// TIA Portal project "Diplomski_rad" (V16)

(* hardware
DEVICE "S7-1200 station_2"  S7-1200 Station
   slot 0: "Rack_0"  S7-1200 Rack  Rack  V1.0
   slot 1: "PLC_1"  CPU 1215C DC/DC/DC  6ES7 215-1AG40-0XB0  V4.4
DEVICE "HMI_1"  KTP700 Basic PN
   slot 0: "HMI_1"  KTP700 Basic PN  6AV2 123-2GB03-0AX0  16.0.0.0
   slot 1: "HMI_RT_1"  KTP700 Basic PN  6AV2 123-2GB03-0AX0  16.0.0.0
   slot 5: "HMI_1.IE_CP_1"  PROFINET Interface  16.0.0.0
      slot 1: "PROFINET Interface_1"  PROFINET Interface
         slot 1: "Port_1"  Port
DEVICE "SCALANCE X005"  SCALANCE X-Station
   slot 0: "SCALANCE X rack"  Rail
   slot 0: "Switch_1"  6GK5 005-0BA00-1AB2  V1.0
DEVICE "GSD device_1"  GSD.Device.PN
   slot 0: "Rack"  Rack  V1.0
   slot 0: "EX260-SPN"  EX260 SPN 1/2  EX260-SPN
      slot 0: "EX260 SPN 1/2"  EX260 SPN 1/2
      slot 1: "Interface"  Interface
         slot 1: "Port 1 - RJ45"  Port 1 - RJ45
         slot 2: "Port 2 - RJ45"  Port 2 - RJ45
      slot 1: "  4 byte  Output_1"    4 byte  Output
         slot 0: "  4 byte  Output"    4 byte  Output
DEVICE "ET 200SP station_1"  ET 200SP-Station
   slot 0: "Rack_0"  Rack  6ES5 710-8MAx1
   slot 0: "IO device_1"  IM 155-6 PN/2 HF  6ES7 155-6AU01-0CN0  V4.2
   slot 1: "DI 8x24VDC HF_1"  DI 8x24VDC HF  6ES7 131-6BF00-0CA0  V2.0
      slot 1: "DI 8x24VDC HF_1"  DI 8x24VDC HF
   slot 2: "DI 8x24VDC HF_2"  DI 8x24VDC HF  6ES7 131-6BF00-0CA0  V2.0
      slot 1: "DI 8x24VDC HF_2"  DI 8x24VDC HF
   slot 3: "DQ 8x24VDC/0.5A HF_1"  DQ 8x24VDC/0.5A HF  6ES7 132-6BF00-0CA0  V2.0
      slot 1: "DQ 8x24VDC/0.5A HF_1"  DQ 8x24VDC/0.5A HF
   slot 4: "DQ 8x24VDC/0.5A HF_2"  DQ 8x24VDC/0.5A HF  6ES7 132-6BF00-0CA0  V2.0
      slot 1: "DQ 8x24VDC/0.5A HF_2"  DQ 8x24VDC/0.5A HF
   slot 5: "AI 4xU/I 2-wire ST_1"  AI 4xU/I 2-wire ST  6ES7 134-6HD01-0BA1  V2.0
      slot 1: "AI 4xU/I 2-wire ST_1"  AI 4xU/I 2-wire ST
   slot 6: "AQ 2xU/I HF_1"  AQ 2xU/I HF  6ES7 135-6HB00-0CA1  V1.0
      slot 1: "AQ 2xU/I HF_1"  AQ 2xU/I HF
   slot 7: "TM Timer DIDQ 10x24V_1"  TM Timer DIDQ 10x24V  6ES7 138-6CG00-0BA0  V1.0
      slot 1: "TM Timer DIDQ 10x24V_1"  TM Timer DIDQ 10x24V
   slot 8: "Server module_1"  Server module  6ES7 193-6PA00-0AA0  V1.1
      slot 1: "Server module_1"  Server module
   slot 127: "BA 2xRJ45"  BA 2xRJ45  6ES7 193-6AR00-0AA0  V0.0
      slot 1: "Port_1"  X1 P1 R  6ES7 193-6AR00-0AA0  V0.0
      slot 2: "Port_2"  X1 P2 R  6ES7 193-6AR00-0AA0  V0.0
*)

// ===== PLC "PLC_1"  CPU 1215C DC/DC/DC =====

VAR_GLOBAL   // PLC tag table "Default tag table"
   "Tag_1" AT %M0.0 : Bool;
   "Tag_2" AT %M0.1 : Bool;
   "Tag_3" AT %M0.2 : Bool;
   "Tag_4" AT %M0.3 : Bool;
   "Tag_5" AT %M0.4 : Bool;
END_VAR

VAR_GLOBAL   // PLC tag table "PLC I/O"
   "izlaz1" AT %Q0.0 : Bool;   // PTO_motor_1
   "izlaz2" AT %Q0.1 : Bool;   // Enable_motor_1
   "izlaz3" AT %Q0.2 : Bool;   // Direction_motor_1
   "izlaz4" AT %Q0.3 : Bool;   // PTO_motor_2
   "izlaz5" AT %Q0.4 : Bool;   // Enable_motor_2
   "izlaz6" AT %Q0.5 : Bool;   // Direction_motor_2
   "izlaz7" AT %Q0.6 : Bool;
   "izlaz8" AT %Q0.7 : Bool;
   "ulaz1" AT %I0.0 : Bool;
   "ulaz2" AT %I0.1 : Bool;
   "ulaz3" AT %I0.2 : Bool;   // Home_vodilica_1_(manja)
   "ulaz4" AT %I0.3 : Bool;   // Home_vodilica_2_(veca)
   "ulaz5" AT %I0.4 : Bool;   // HW_limiter_0_vodilica_1
   "ulaz6" AT %I0.5 : Bool;   // HW_limiter_1_vodilica_1
   "ulaz7" AT %I0.6 : Bool;   // HW_limiter_0_vodilica_2
   "ulaz8" AT %I0.7 : Bool;   // HW_limiter_1_vodilica_2
END_VAR

VAR_GLOBAL   // PLC tag table "Distro I/O"
   "Dist_ulaz1" AT %I2.0 : Bool;
   "Dist_ulaz2" AT %I2.1 : Bool;
   "Dist_ulaz3" AT %I2.2 : Bool;
   "Dist_ulaz4" AT %I2.3 : Bool;
   "Dist_ulaz5" AT %I2.4 : Bool;   // Senzor_cilindar_uvučen
   "Dist_ulaz6" AT %I2.5 : Bool;   // Senzor_cilindar_izvučen
   "Dist_ulaz7" AT %I2.6 : Bool;   // Senzor_hvataljka_otvorena
   "Dist_ulaz8" AT %I2.7 : Bool;   // Senzor_hvataljka_zatvorena
   "Dist_izlaz1" AT %Q2.0 : Bool;
   "Dist_izlaz2" AT %Q2.1 : Bool;
   "Dist_izlaz3" AT %Q2.2 : Bool;
   "Dist_izlaz4" AT %Q2.3 : Bool;
   "Dist_izlaz5" AT %Q2.4 : Bool;
   "Dist_izlaz6" AT %Q2.5 : Bool;
   "Dist_izlaz7" AT %Q2.6 : Bool;
   "Dist_izlaz8" AT %Q2.7 : Bool;
END_VAR

VAR_GLOBAL   // PLC tag table "Ventili I/O"
   "Ventil_izlaz_1" AT %Q4.0 : Bool;
   "Ventil_izlaz_2" AT %Q4.1 : Bool;
   "Ventil_izlaz_3" AT %Q4.2 : Bool;
   "Ventil_izlaz_4" AT %Q4.3 : Bool;
   "Otvorena_hvataljka" AT %Q4.4 : Bool;
   "Zatvorena_hvataljka" AT %Q4.5 : Bool;
   "Izvučeni_cilindar" AT %Q4.6 : Bool;
   "Uvučeni_cilindar" AT %Q4.7 : Bool;
   "Ventil_izlaz_9" AT %Q5.0 : Bool;
   "Ventil_izlaz_10" AT %Q5.1 : Bool;
   "Ventil_izlaz_11" AT %Q5.2 : Bool;
   "Ventil_izlaz_12" AT %Q5.3 : Bool;
   "Ventil_izlaz_13" AT %Q5.4 : Bool;
   "Ventil_izlaz_14" AT %Q5.5 : Bool;
   "Ventil_izlaz_15" AT %Q5.6 : Bool;
   "Ventil_izlaz_16" AT %Q5.7 : Bool;
   "Ventil_izlaz_17" AT %Q6.0 : Bool;
   "Ventil_izlaz_18" AT %Q6.1 : Bool;
   "Ventil_izlaz_19" AT %Q6.2 : Bool;
   "Ventil_izlaz_20" AT %Q6.3 : Bool;
   "Ventil_izlaz_21" AT %Q6.4 : Bool;
   "Ventil_izlaz_22" AT %Q6.5 : Bool;
   "Ventil_izlaz_23" AT %Q6.6 : Bool;
   "Ventil_izlaz_24" AT %Q6.7 : Bool;
   "Ventil_izlaz_25" AT %Q7.0 : Bool;
   "Ventil_izlaz_26" AT %Q7.1 : Bool;
   "Ventil_izlaz_27" AT %Q7.2 : Bool;
   "Ventil_izlaz_28" AT %Q7.3 : Bool;
   "Ventil_izlaz_29" AT %Q7.4 : Bool;
   "Ventil_izlaz_30" AT %Q7.5 : Bool;
   "Ventil_izlaz_31" AT %Q7.6 : Bool;
   "Ventil_izlaz_32" AT %Q7.7 : Bool;
END_VAR

TYPE "Motor"
   STRUCT
      Uključi_motor : Bool;
      "Potvrdi_error(reset)" : Bool;
      Pokreni_homing : Bool;
      Pokreni_zaustavljanje : Bool;
      Pokreni_izvršavanje_pomaka_apsolutno : Bool;
      Pokreni_izvršavanje_pomaka_relativno : Bool;
      Željena_pozicija : Real;
      Željeni_pomak : Real;
      Trenutna_pozicija : Real;
      Power_Status : Bool;
      Power_Error : Bool;
      "Potvrdi_error(reset)_Izvršeno" : Bool;
      "Potvrdi_error(reset)_Error" : Bool;
      Home_Izvršeno : Bool;
      Home_izvršeno_barem_jednom : Bool;
      Home_Izvršavanje : Bool;
      Home_Error : Bool;
      Halt_Izvršeno : Bool;
      Halt_Error : Bool;
      Pomak_Apsolutno_Izvršeno : Bool;
      Pomak_Apsolutno_U_Tijeku : Bool;
      Pomak_Apsolutno_Error : Bool;
      Pomak_Relativno_izvršeno : Bool;
      Pomak_Relativno_Error : Bool;
      Brzina_Izvršavanje : Bool;
      Brzina_Error : Bool;
   END_STRUCT;
END_TYPE

DATA_BLOCK "Motor_DB"   // DB2
{ S7_Optimized_Access := 'TRUE' }
VERSION : 0.1
   VAR
      "Motor_1_x-os" : "Motor";
      "Motor_2_y-os" : "Motor";
   END_VAR
BEGIN
END_DATA_BLOCK

DATA_BLOCK "Rucno_upravljanje"   // DB3
{ S7_Optimized_Access := 'TRUE' }
VERSION : 0.1
   VAR
      GORE : Bool;
      DOLJE : Bool;
      LIJEVO : Bool;
      DESNO : Bool;
      GD_izvrsavanje : Bool;
      LD_izvrsavanje : Bool;
      GD_brzina : Real := 12.0;
      LD_brzina : Real := 12.0;
   END_VAR
BEGIN
END_DATA_BLOCK

DATA_BLOCK "Pneumatske_komponente"   // DB5
{ S7_Optimized_Access := 'TRUE' }
VERSION : 0.1
   VAR
      Aktivacija_cilindra : Bool;
      Aktivacija_hvataljke : Bool;
   END_VAR
BEGIN
END_DATA_BLOCK

DATA_BLOCK "Paletizacija_DB"   // DB6
{ S7_Optimized_Access := 'TRUE' }
VERSION : 0.1
// stored: InstanceOfName Paletizacija
"Paletizacija"
BEGIN
END_DATA_BLOCK

DATA_BLOCK "Automatsko_upravljanje"   // DB7
{ S7_Optimized_Access := 'TRUE' }
VERSION : 0.1
   VAR
      Automatski_režim : Bool;
      Paletizacija : Bool;
      Kraj_paletizacije : Bool;
      Broj_komada_palete_x : Int := 2;
      Broj_komada_palete_y : Int := 2;
      Pauza : Bool;
      Lokalizacija_objekata_i_sortiranje : Bool;
      Lokalizacija_objekata_x_koordinata : Real;
      Lokalizacija_objekata_y_koordinata : Real;
      Primljeni_podatci : Bool;
      Lokalizacija_objekata_boja : Int;
      Zahtjev_za_poziciju : Bool;
   END_VAR
BEGIN
END_DATA_BLOCK

DATA_BLOCK "Vizija_python"   // DB10
{ S7_Optimized_Access := 'FALSE' }
VERSION : 0.1
   VAR
      Slanje_podataka : Byte;
      Slanje_podataka_stanje : Bool;
      Primanje_podataka : Char;
      Broj_primljenih_podataka : Int := 0;
      Primljeno : Bool;
      Broj : DInt;
      X_koordinata : DInt := 0;
      Y_koordinata : DInt := 0;
      Boja : DInt := 0;
      Broj_razmaka : DInt := 0;
      "Koeficijent_px/mm_x" : Real := 4.9;
      "Koeficijent_px/mm_y" : Real := 4.85;
      Offset_k_s_kamere_x : Real := 0.0;
      Offset_k_s_kamere_y : Real := 47.0;
   END_VAR
BEGIN
END_DATA_BLOCK

DATA_BLOCK "Lokalizacija_objekata_i_sortiranje_DB"   // DB13
{ S7_Optimized_Access := 'TRUE' }
VERSION : 0.1
// stored: InstanceOfName Lokalizacija_objekata_i_sortiranje
"Lokalizacija_objekata_i_sortiranje"
BEGIN
END_DATA_BLOCK

DATA_BLOCK "Motor_upravljanje_DB"   // DB17
{ S7_Optimized_Access := 'TRUE' }
VERSION : 0.1
// stored: InstanceOfName Motor_upravljanje
"Motor_upravljanje"
BEGIN
END_DATA_BLOCK

DATA_BLOCK "Motor_upravljanje_DB_2"   // DB18
{ S7_Optimized_Access := 'TRUE' }
VERSION : 0.1
// stored: InstanceOfName Motor_upravljanje
"Motor_upravljanje"
BEGIN
END_DATA_BLOCK

// folder: System blocks/Program resources

DATA_BLOCK "PLC_1_TCP_DB"   // DB9
{ S7_Optimized_Access := 'TRUE' }
AUTHOR : SIMATIC
FAMILY : MC7Plus
NAME : TC_IP_v4
VERSION : 1.0
// stored: InstanceOfName TCON_IP_v4
"TCON_IP_v4"
BEGIN
   ID := 1;
   InterfaceId := 64;
   LocalPort := 2000;
END_DATA_BLOCK

DATA_BLOCK "Tajmer_za_slanje_poruke"   // DB12
{ S7_Optimized_Access := 'TRUE' }
AUTHOR : Simatic
FAMILY : IEC
NAME : IEC_TMR
VERSION : 1.0
// stored: InstanceOfName IEC_TIMER
"IEC_TIMER"
BEGIN
END_DATA_BLOCK

DATA_BLOCK "IEC_Timer_0_DB_1"   // DB14
{ S7_Optimized_Access := 'TRUE' }
AUTHOR : Simatic
FAMILY : IEC
NAME : IEC_TMR
VERSION : 1.0
// stored: InstanceOfName IEC_TIMER
"IEC_TIMER"
BEGIN
END_DATA_BLOCK

DATA_BLOCK "Tajmer_za_primanje_poruke"   // DB15
{ S7_Optimized_Access := 'TRUE' }
AUTHOR : Simatic
FAMILY : IEC
NAME : IEC_TMR
VERSION : 1.0
// stored: InstanceOfName IEC_TIMER
"IEC_TIMER"
BEGIN
END_DATA_BLOCK

// folder: (top level)

DATA_BLOCK "Axis_1"   // DB1, Motion_DB
{ S7_Optimized_Access := 'TRUE' }
AUTHOR : SIMATIC
FAMILY : BasicMC
NAME : TO_PosAx
VERSION : 7.0
// stored: InstanceOfName TO_PositioningAxis
"TO_PositioningAxis"
BEGIN
   // Axis.DirectionOutputEnabledCU = TRUE
   // Axis.PositionLimitsMax_AddressCU = %I0.5
   // Axis.PositionLimitsMin_AddressCU = %I0.4
   // Axis.PassiveHomingReferencePointSwitch_AddressCU = %I0.2
   // Axis.HomingReferencePointSwitch_AddressCU = %I0.2
   // Axis.LengthUnitNormalized.Distance = 1013
   // Axis.EnableOutput_AddressCU = %Q0.1
   // Axis.OnlinePtoModeCU = 16#0000_0002
   // Axis.SelectedChannel2EnumCU = %Q0.2
   // Axis.SelectedChannel1EnumCU = %Q0.0
   // Pulse.MinDeltaDeltaFrequencyCU = 0.004
   // Pulse.MaxDeltaDeltaFrequencyCU = 1.0E+10
   // Pulse.MinDeltaFrequencyCU = 0.005
   // Pulse.MaxDeltaFrequencyCU = 9.5E+9
   // Pulse.MinFrequencyCU = 1.0
   // Pulse.MaxFrequencyCU = 100000.0
   // Pulse.OutputSourceCU = 16#0000_0000
   // Axis.SelectPTO = 0
END_DATA_BLOCK

DATA_BLOCK "Axis_2"   // DB4, Motion_DB
{ S7_Optimized_Access := 'TRUE' }
AUTHOR : SIMATIC
FAMILY : BasicMC
NAME : TO_PosAx
VERSION : 7.0
// stored: InstanceOfName TO_PositioningAxis
"TO_PositioningAxis"
BEGIN
   // Axis.PositionLimitsMax_AddressCU = %I0.7
   // Axis.PositionLimitsMin_AddressCU = %I0.6
   // Axis.PassiveHomingReferencePointSwitch_AddressCU = %I0.3
   // Axis.HomingReferencePointSwitch_AddressCU = %I0.3
   // Axis.LengthUnitNormalized.Distance = 1013
   // Axis.EnableOutput_AddressCU = %Q0.4
   // Axis.OnlinePtoModeCU = 16#0000_0002
   // Axis.DirectionOutputEnabledCU = TRUE
   // Axis.SelectedChannel2EnumCU = %Q0.5
   // Axis.SelectedChannel1EnumCU = %Q0.3
   // Pulse.MinDeltaDeltaFrequencyCU = 0.004
   // Pulse.MaxDeltaDeltaFrequencyCU = 1.0E+10
   // Pulse.MinDeltaFrequencyCU = 0.005
   // Pulse.MaxDeltaFrequencyCU = 9.5E+9
   // Pulse.MinFrequencyCU = 1.0
   // Pulse.MaxFrequencyCU = 100000.0
   // Pulse.OutputSourceCU = 16#0000_0000
   // Axis.SelectPTO = 1
   // Axis.OnlinePtoIndexCU = 1
END_DATA_BLOCK

FUNCTION_BLOCK "Motor_upravljanje"   // FB1, LAD
{ S7_Optimized_Access := 'TRUE' }
VERSION : 0.1
   VAR_INPUT
      Os : TO_PositioningAxis;
      Uključi_motor : Bool;
      "Potvrdi_error(reset)" : Bool;
      Pokreni_homing : Bool;
      Pokreni_zaustavljanje : Bool;
      Pokreni_izvršavanje_pomaka_apsolutno : Bool;
      Pokreni_izvršavanje_pomaka_relativno : Bool;
      Željena_pozicija : Real;
      Željeni_pomak : Real;
      Izvršavanje_direktno_preko_gumba : Bool;
      Maks_brzina_izvršavanje_preko_gumba : Real;
      Gumb_od_motora : Bool;
      Gumb_prema_motoru : Bool;
   END_VAR
   VAR_OUTPUT
      Trenutna_pozicija : Real;
      Power_Status : Bool;
      Power_Error : Bool;
      "Potvrdi_error(reset)_Izvršeno" : Bool;
      "Potvrdi_error(reset)_Error" : Bool;
      Home_Izvršeno : Bool;
      Home_izvršeno_barem_jednom : Bool;
      Home_izvršavanje : Bool;
      Home_Error : Bool;
      Halt_Izvršeno : Bool;
      Halt_Error : Bool;
      Pomak_Apsolutno_Izvršeno : Bool;
      Pomak_Apsolutno_U_Tijeku : Bool;
      Pomak_Apsolutno_Error : Bool;
      Pomak_Relativno_Izvršeno : Bool;
      Pomak_Relativno_Error : Bool;
      Brzina_Izvršavanje : Bool;
      Brzina_Error : Bool;
   END_VAR
   VAR
      MC_Power_Instance : MC_Power;
      MC_Reset_Instance : MC_Reset;
      MC_Home_Instance : MC_Home;
      MC_Halt_Instance : MC_Halt;
      MC_MoveAbsolute_Instance : MC_MoveAbsolute;
      MC_MoveRelative_Instance : MC_MoveRelative;
      MC_MoveVelocity_Instance : MC_MoveVelocity;
      Provjera_edga : Bool;
   END_VAR
   VAR_TEMP   // added for the SCL form of the ladder/FBD networks
      _w1 : Bool;
   END_VAR
BEGIN

REGION Network 1
   // MC_Power - Uključuje motor, bez njega se ne može pokrenuti
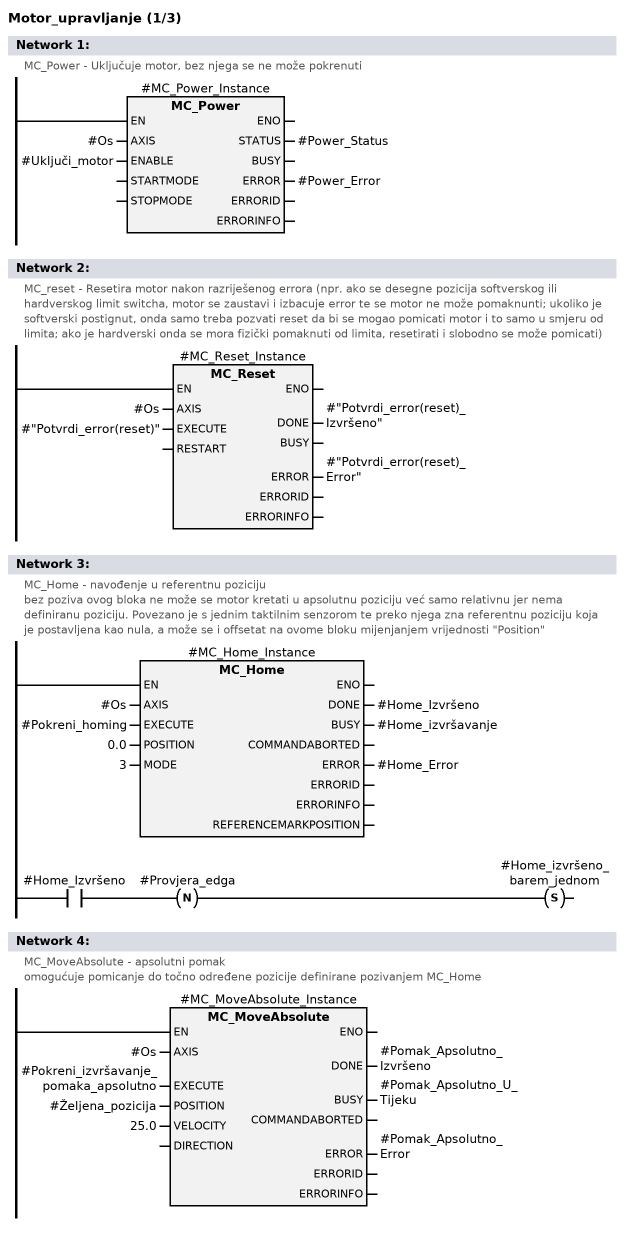
   #MC_Power_Instance(Axis := #Os, Enable := #Uključi_motor, Status => #Power_Status, Error => #Power_Error);   // MC_Power
END_REGION

REGION Network 2
   // MC_reset - Resetira motor nakon razriješenog errora (npr. ako se desegne pozicija softverskog ili hardverskog limit switcha, motor se zaustavi i izbacuje error te se motor ne može pomaknunti; ukoliko je softverski postignut, onda samo treba pozvati reset da bi se mogao pomicati motor i to samo u smjeru od limita; ako je hardverski onda se mora fizički pomaknuti od limita, resetirati i slobodno se može pomicati)
   #MC_Reset_Instance(Axis := #Os,   // MC_Reset
                      Execute := #"Potvrdi_error(reset)",
                      Done => #"Potvrdi_error(reset)_Izvršeno",
                      Error => #"Potvrdi_error(reset)_Error");
END_REGION

REGION Network 3
   // MC_Home - navođenje u referentnu poziciju
   // bez poziva ovog bloka ne može se motor kretati u apsolutnu poziciju već samo relativnu jer nema definiranu poziciju. Povezano je s jednim taktilnim senzorom te preko njega zna referentnu poziciju koja je postavljena kao nula, a može se i offsetat na ovome bloku mijenjanjem vrijednosti "Position"
   #MC_Home_Instance(Axis := #Os,   // MC_Home
                     Execute := #Pokreni_homing,
                     Position := 0.0,
                     Mode := 3,
                     Done => #Home_Izvršeno,
                     Busy => #Home_izvršavanje,
                     Error => #Home_Error);
   #_w1 := NOT #Home_Izvršeno AND #Provjera_edga;   // falling edge
   #Provjera_edga := #Home_Izvršeno;
   IF #_w1 THEN #Home_izvršeno_barem_jednom := TRUE; END_IF;
END_REGION

REGION Network 4
   // MC_MoveAbsolute - apsolutni pomak
   // omogućuje pomicanje do točno određene pozicije definirane pozivanjem MC_Home
   #MC_MoveAbsolute_Instance(Axis := #Os,   // MC_MoveAbsolute
                           Execute := #Pokreni_izvršavanje_pomaka_apsolutno,
                           Position := #Željena_pozicija,
                           Velocity := 25.0,
                           Done => #Pomak_Apsolutno_Izvršeno,
                           Busy => #Pomak_Apsolutno_U_Tijeku,
                           Error => #Pomak_Apsolutno_Error);
END_REGION

REGION Network 5
   // MC_MoveRelative - relativni pomak
   // omogućuje pomicanje za točno određenu udaljenost
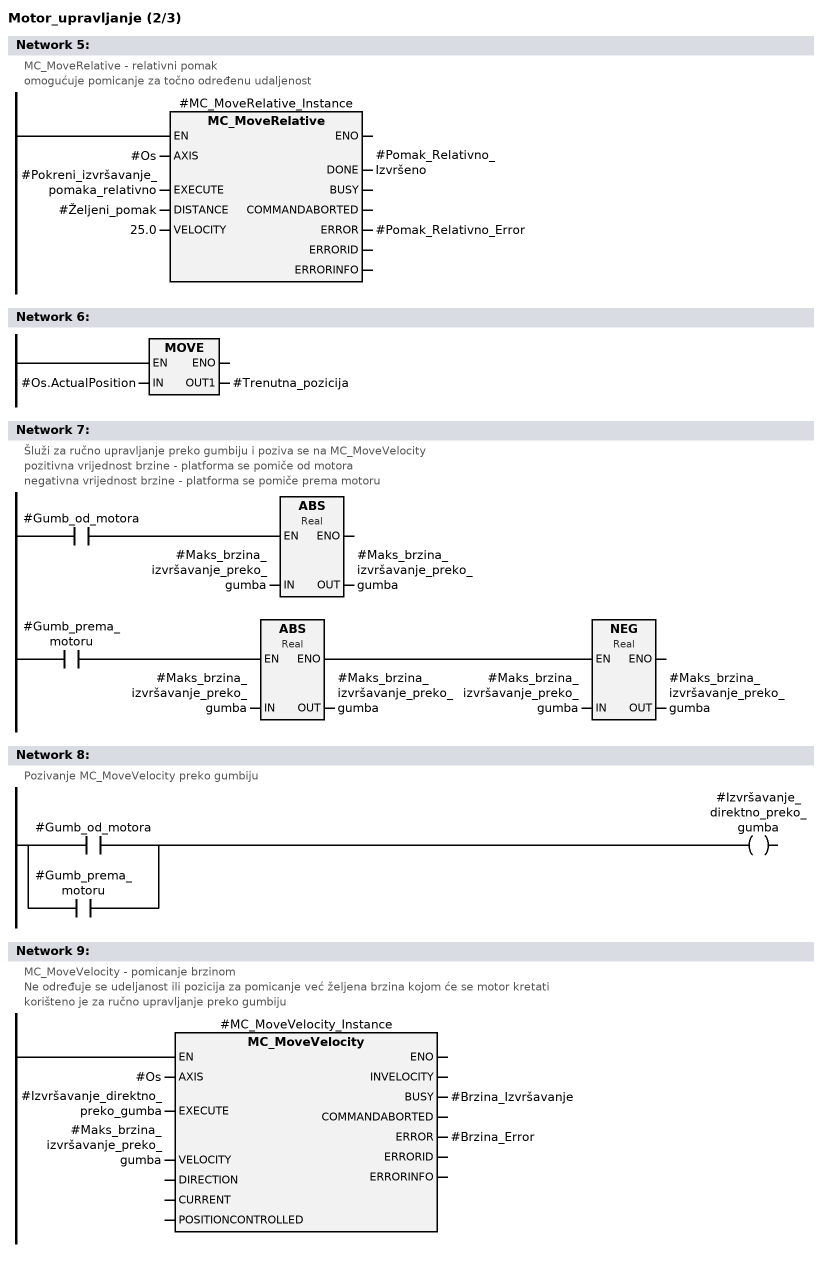
   #MC_MoveRelative_Instance(Axis := #Os,   // MC_MoveRelative
                           Execute := #Pokreni_izvršavanje_pomaka_relativno,
                           Distance := #Željeni_pomak,
                           Velocity := 25.0,
                           Done => #Pomak_Relativno_Izvršeno,
                           Error => #Pomak_Relativno_Error);
END_REGION

REGION Network 6
   RUNG wire#powerrail
      Move(in := #Os.ActualPosition, out1 => #Trenutna_pozicija)
   END_RUNG
   // the same network as SCL:
   #Trenutna_pozicija := #Os.ActualPosition;
END_REGION

REGION Network 7
   // Šluži za ručno upravljanje preko gumbiju i poziva se na MC_MoveVelocity 
   // pozitivna vrijednost brzine - platforma se pomiče od motora
   // negativna vrijednost brzine - platforma se pomiče prema motoru
   RUNG wire#powerrail
      Contact( #Gumb_od_motora )
      { S7_Templates := "SrcType := Real" } Abs(in := #Maks_brzina_izvršavanje_preko_gumba, out => #Maks_brzina_izvršavanje_preko_gumba)
   END_RUNG
   RUNG wire#powerrail
      Contact( #Gumb_prema_motoru )
      { S7_Templates := "SrcType := Real" } Abs(in := #Maks_brzina_izvršavanje_preko_gumba, out => #Maks_brzina_izvršavanje_preko_gumba)
      { S7_Templates := "SrcType := Real"; S7_GenerateENO := "TRUE" } Neg(in := #Maks_brzina_izvršavanje_preko_gumba, out => #Maks_brzina_izvršavanje_preko_gumba)
   END_RUNG
   // the same network as SCL:
   IF #Gumb_od_motora THEN
       #Maks_brzina_izvršavanje_preko_gumba := ABS(#Maks_brzina_izvršavanje_preko_gumba);
   END_IF;
   IF #Gumb_prema_motoru THEN
       #Maks_brzina_izvršavanje_preko_gumba := ABS(#Maks_brzina_izvršavanje_preko_gumba);
       #Maks_brzina_izvršavanje_preko_gumba := -#Maks_brzina_izvršavanje_preko_gumba;
   END_IF;
END_REGION

REGION Network 8
   // Pozivanje MC_MoveVelocity preko gumbiju
   RUNG wire#powerrail
      Contact( #Gumb_od_motora )
      wire#w1
      Coil( #Izvršavanje_direktno_preko_gumba )
   END_RUNG
   RUNG wire#powerrail
      Contact( #Gumb_prema_motoru )
   END_RUNG wire#w1
   // the same network as SCL:
   #Izvršavanje_direktno_preko_gumba := #Gumb_od_motora OR #Gumb_prema_motoru;
END_REGION

REGION Network 9
   // MC_MoveVelocity - pomicanje brzinom
   // Ne određuje se udeljanost ili pozicija za pomicanje već željena brzina kojom će se motor kretati
   // korišteno je za ručno upravljanje preko gumbiju
   #MC_MoveVelocity_Instance(Axis := #Os,   // MC_MoveVelocity
                           Execute := #Izvršavanje_direktno_preko_gumba,
                           Velocity := #Maks_brzina_izvršavanje_preko_gumba,
                           Busy => #Brzina_Izvršavanje,
                           Error => #Brzina_Error);
END_REGION

REGION Network 10
   // MC_Halt - zaustavljanje
   // služi za zaustavljanje kretnje motora, bilo u navođenju u nulu, pozicijsko ili brzinsko
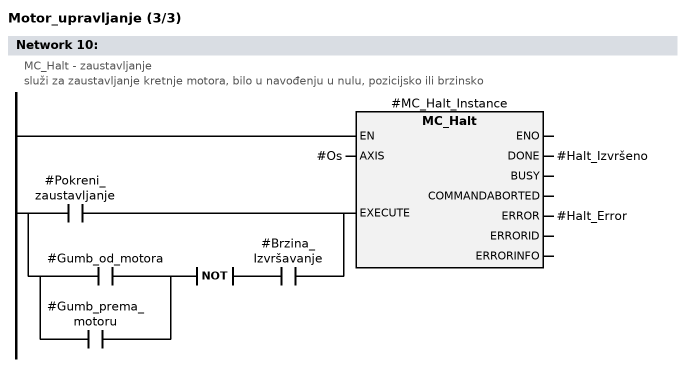
   #MC_Halt_Instance(Axis := #Os,   // MC_Halt
                     Execute := #Pokreni_zaustavljanje OR (NOT (#Gumb_od_motora OR #Gumb_prema_motoru) AND #Brzina_Izvršavanje),
                     Done => #Halt_Izvršeno,
                     Error => #Halt_Error);
END_REGION
END_FUNCTION_BLOCK

FUNCTION_BLOCK "Lokalizacija_objekata_i_sortiranje"   // FB2, LAD
{ S7_Optimized_Access := 'TRUE' }
VERSION : 0.1
   VAR_INPUT
      Senzor_cilindar_uvučen : Bool;
      Senzor_cilindar_izvučen : Bool;
      Senzor_hvataljka_zatvorena : Bool;
      Senzor_hvataljka_otvorena : Bool;
      Home_izvršeno_x : Bool;
      Home_izvršeno_y : Bool;
      Trenutna_pozicija_x : Real;
      Trenutna_pozicija_y : Real;
      Pomak_izvršen_x : Bool;
      Pomak_izvršen_y : Bool;
      Dobivena_pozicija_x : Real;
      Dobivena_pozicija_y : Real;
      Dobivena_boja : Int;
      Pauza : Bool;
   END_VAR
   VAR_OUTPUT
      Aktivacija_cilindra : Bool;   // 1 - izvučen, 0 - uvučen
      Aktivacija_hvataljke : Bool;   // 1 - zatvorena, 0 - otvorena
      Home_x : Bool;
      Home_y : Bool;
      Željeni_apsolutni_pomak_x : Real;
      Željeni_apsolutni_pomak_y : Real;
      Izvršavanje_pomaka_x : Bool;
      Izvršavanje_pomaka_y : Bool;
      Zaustavljanje_x : Bool;
      Zaustavljanje_y : Bool;
   END_VAR
   VAR_IN_OUT
      Poziv_lokalizacija_objekata_i_sortiranje : Bool;
      Zahtjev_za_poziciju : Bool;
      Dobiveni_podaci_predmeta : Bool;
   END_VAR
   VAR
      Poziv_inicijalizacija : Bool;   // Oznaka pozivanja inicijalizacije
      Provjera_kraja_inicijalizacije : Bool;
      Provjera_poziva_lokalizacije_objekata_i_sortiranja : Bool;
      Proces_kretanja : Bool;   // Proces kretnje platforme
      Provjera_procesa_kretanja : Bool;
      Provjera_zahtjeva_za_poziciju : Bool;
      Provjera_kraja_pneumatike : Bool;
      Brojac : Int;
      Brojac_MOD : Int;
      Zaustavljen_x : Bool;
      Zaustavljen_y : Bool;
      Kraj_pneumatike : Bool;   // Izvršavanje koraka pneumatike je gotovo
      Prolaz_hvataljke : Bool;   // Provjera je li hvataljka bila aktivirana tijekom koraka pneumatike, bez ove varijable bila bi dva identična pozivanja pa se nebi znalo ima li hvataljka uhvaćen predmet ili ne
      Provjera_uvlačenja_cilindra : Bool;
      Provjera_zaustavljanja : Bool;
      Provjera_pauze : Bool;
   END_VAR
   VAR_TEMP
      Pomicanje_homiranje_x : Bool;
      Pomicanje_homiranje_y : Bool;
      Cilindar_je_uvucen : Bool;
      Hvataljka_je_otvorena : Bool;
   END_VAR
   VAR_TEMP   // added for the SCL form of the ladder/FBD networks
      _w1 : Bool;
      _w2 : Bool;
      _w3 : Bool;
      _w4 : Bool;
   END_VAR
BEGIN

REGION Network 1: Oznaka pozivanja inicijalizacije
   // Inicijalizacija manipulatora
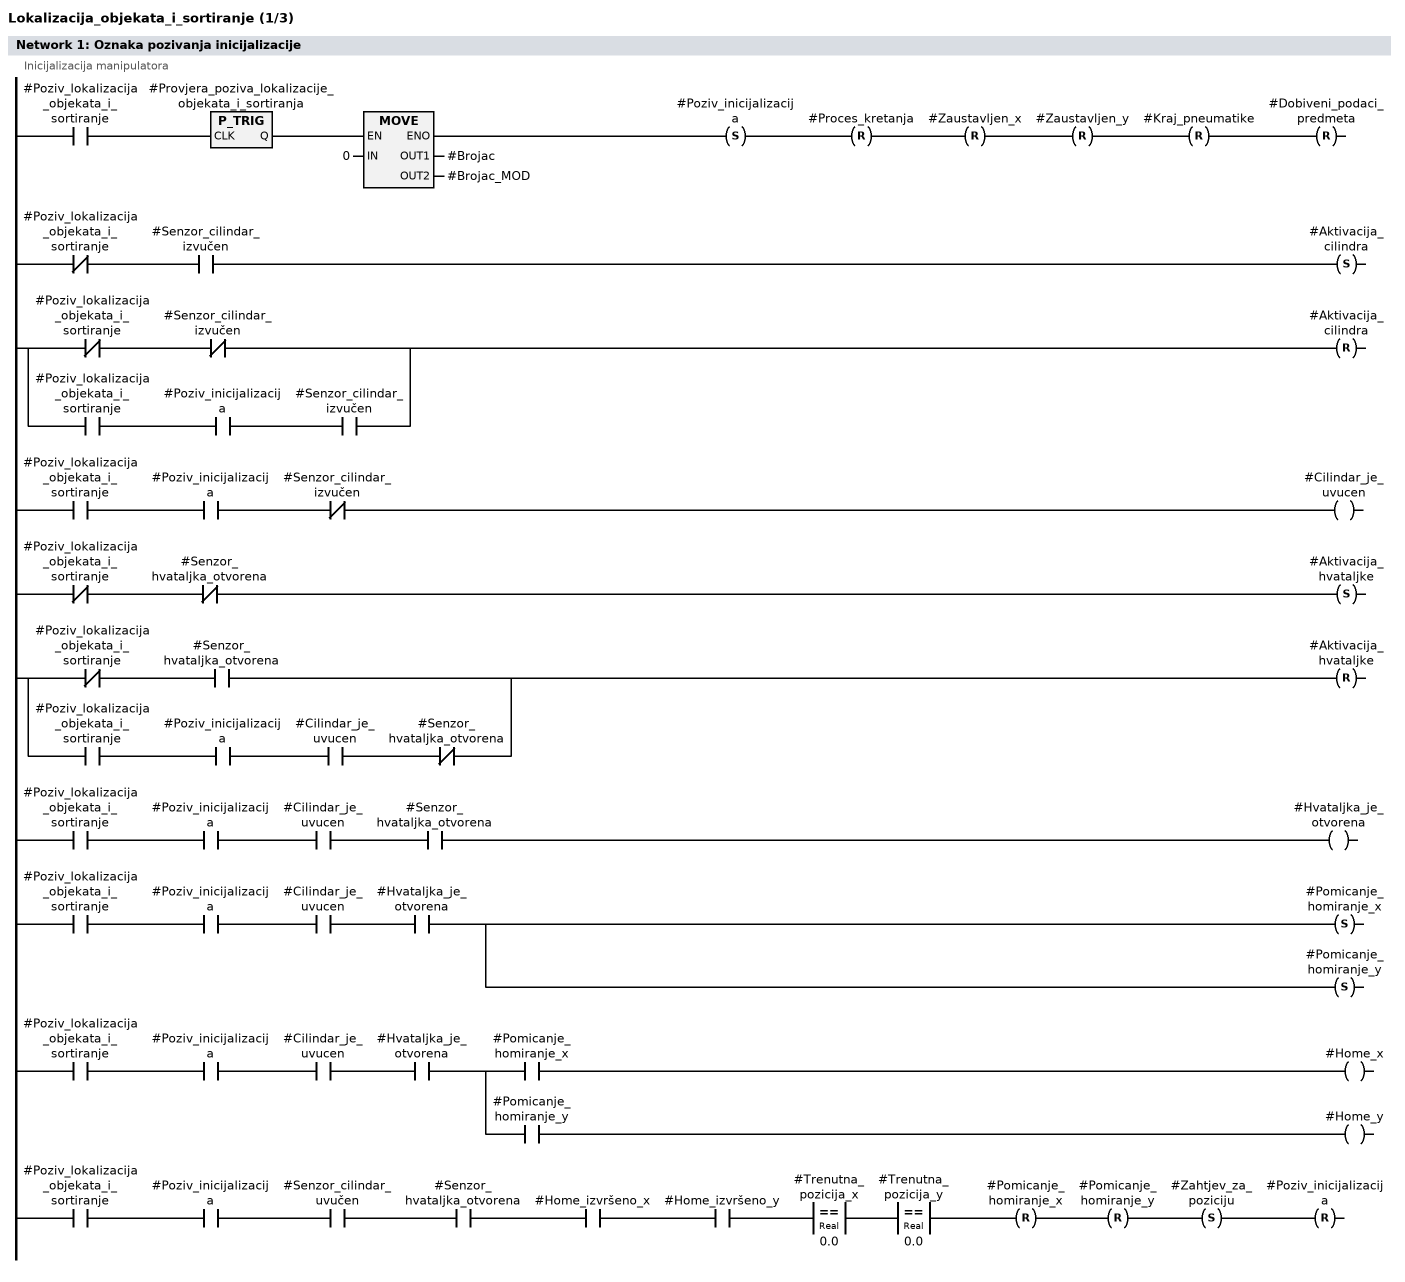
   RUNG wire#powerrail
      Contact( #Poziv_lokalizacija_objekata_i_sortiranje )
      P_Trig( #Provjera_poziva_lokalizacije_objekata_i_sortiranja )
      Move(in := 0, out1 => #Brojac, out2 => #Brojac_MOD)
      S_Coil( #Poziv_inicijalizacija )
      R_Coil( #Proces_kretanja )
      R_Coil( #Zaustavljen_x )
      R_Coil( #Zaustavljen_y )
      R_Coil( #Kraj_pneumatike )
      R_Coil( #Dobiveni_podaci_predmeta )
   END_RUNG
   RUNG wire#powerrail
      I_Contact( #Poziv_lokalizacija_objekata_i_sortiranje )
      Contact( #Senzor_cilindar_izvučen )
      S_Coil( #Aktivacija_cilindra )
   END_RUNG
   RUNG wire#powerrail
      I_Contact( #Poziv_lokalizacija_objekata_i_sortiranje )
      I_Contact( #Senzor_cilindar_izvučen )
      wire#w1
      R_Coil( #Aktivacija_cilindra )
   END_RUNG
   RUNG wire#powerrail
      Contact( #Poziv_lokalizacija_objekata_i_sortiranje )
      Contact( #Poziv_inicijalizacija )
      Contact( #Senzor_cilindar_izvučen )
   END_RUNG wire#w1
   RUNG wire#powerrail
      Contact( #Poziv_lokalizacija_objekata_i_sortiranje )
      Contact( #Poziv_inicijalizacija )
      I_Contact( #Senzor_cilindar_izvučen )
      Coil( #Cilindar_je_uvucen )
   END_RUNG
   RUNG wire#powerrail
      I_Contact( #Poziv_lokalizacija_objekata_i_sortiranje )
      I_Contact( #Senzor_hvataljka_otvorena )
      S_Coil( #Aktivacija_hvataljke )
   END_RUNG
   RUNG wire#powerrail
      I_Contact( #Poziv_lokalizacija_objekata_i_sortiranje )
      Contact( #Senzor_hvataljka_otvorena )
      wire#w2
      R_Coil( #Aktivacija_hvataljke )
   END_RUNG
   RUNG wire#powerrail
      Contact( #Poziv_lokalizacija_objekata_i_sortiranje )
      Contact( #Poziv_inicijalizacija )
      Contact( #Cilindar_je_uvucen )
      I_Contact( #Senzor_hvataljka_otvorena )
   END_RUNG wire#w2
   RUNG wire#powerrail
      Contact( #Poziv_lokalizacija_objekata_i_sortiranje )
      Contact( #Poziv_inicijalizacija )
      Contact( #Cilindar_je_uvucen )
      Contact( #Senzor_hvataljka_otvorena )
      Coil( #Hvataljka_je_otvorena )
   END_RUNG
   RUNG wire#powerrail
      Contact( #Poziv_lokalizacija_objekata_i_sortiranje )
      Contact( #Poziv_inicijalizacija )
      Contact( #Cilindar_je_uvucen )
      Contact( #Hvataljka_je_otvorena )
      wire#w3
      S_Coil( #Pomicanje_homiranje_x )
   END_RUNG
   RUNG wire#w3
      S_Coil( #Pomicanje_homiranje_y )
   END_RUNG
   RUNG wire#powerrail
      Contact( #Poziv_lokalizacija_objekata_i_sortiranje )
      Contact( #Poziv_inicijalizacija )
      Contact( #Cilindar_je_uvucen )
      Contact( #Hvataljka_je_otvorena )
      wire#w4
      Contact( #Pomicanje_homiranje_x )
      Coil( #Home_x )
   END_RUNG
   RUNG wire#w4
      Contact( #Pomicanje_homiranje_y )
      Coil( #Home_y )
   END_RUNG
   RUNG wire#powerrail
      Contact( #Poziv_lokalizacija_objekata_i_sortiranje )
      Contact( #Poziv_inicijalizacija )
      Contact( #Senzor_cilindar_uvučen )
      Contact( #Senzor_hvataljka_otvorena )
      Contact( #Home_izvršeno_x )
      Contact( #Home_izvršeno_y )
      { S7_Templates := "SrcType := Real" } EQ_Contact(in1 := #Trenutna_pozicija_x, in2 := 0.0)
      { S7_Templates := "SrcType := Real" } EQ_Contact(in1 := #Trenutna_pozicija_y, in2 := 0.0)
      R_Coil( #Pomicanje_homiranje_x )
      R_Coil( #Pomicanje_homiranje_y )
      S_Coil( #Zahtjev_za_poziciju )
      R_Coil( #Poziv_inicijalizacija )
   END_RUNG
   // the same network as SCL:
   #_w1 := #Poziv_lokalizacija_objekata_i_sortiranje AND NOT #Provjera_poziva_lokalizacije_objekata_i_sortiranja;   // rising edge
   #Provjera_poziva_lokalizacije_objekata_i_sortiranja := #Poziv_lokalizacija_objekata_i_sortiranje;
   IF #_w1 THEN
       #Brojac := 0;
       #Brojac_MOD := 0;
       #Poziv_inicijalizacija := TRUE;
       #Proces_kretanja := FALSE;
       #Zaustavljen_x := FALSE;
       #Zaustavljen_y := FALSE;
       #Kraj_pneumatike := FALSE;
       #Dobiveni_podaci_predmeta := FALSE;
   END_IF;
   IF NOT #Poziv_lokalizacija_objekata_i_sortiranje AND #Senzor_cilindar_izvučen THEN
       #Aktivacija_cilindra := TRUE;
   END_IF;
   IF (NOT #Poziv_lokalizacija_objekata_i_sortiranje AND NOT #Senzor_cilindar_izvučen) OR (#Poziv_lokalizacija_objekata_i_sortiranje AND #Poziv_inicijalizacija AND #Senzor_cilindar_izvučen) THEN
       #Aktivacija_cilindra := FALSE;
   END_IF;
   #Cilindar_je_uvucen := #Poziv_lokalizacija_objekata_i_sortiranje AND #Poziv_inicijalizacija AND NOT #Senzor_cilindar_izvučen;
   IF NOT #Poziv_lokalizacija_objekata_i_sortiranje AND NOT #Senzor_hvataljka_otvorena THEN
       #Aktivacija_hvataljke := TRUE;
   END_IF;
   IF (NOT #Poziv_lokalizacija_objekata_i_sortiranje AND #Senzor_hvataljka_otvorena) OR (#Poziv_lokalizacija_objekata_i_sortiranje AND #Poziv_inicijalizacija AND #Cilindar_je_uvucen AND NOT #Senzor_hvataljka_otvorena) THEN
       #Aktivacija_hvataljke := FALSE;
   END_IF;
   #Hvataljka_je_otvorena := #Poziv_lokalizacija_objekata_i_sortiranje AND #Poziv_inicijalizacija AND #Cilindar_je_uvucen AND #Senzor_hvataljka_otvorena;
   IF #Poziv_lokalizacija_objekata_i_sortiranje AND #Poziv_inicijalizacija AND #Cilindar_je_uvucen AND #Hvataljka_je_otvorena THEN
       #Pomicanje_homiranje_x := TRUE;
       #Pomicanje_homiranje_y := TRUE;
   END_IF;
   #_w2 := #Poziv_lokalizacija_objekata_i_sortiranje AND #Poziv_inicijalizacija AND #Cilindar_je_uvucen AND #Hvataljka_je_otvorena;
   #Home_x := #_w2 AND #Pomicanje_homiranje_x;
   #Home_y := #_w2 AND #Pomicanje_homiranje_y;
   IF #Poziv_lokalizacija_objekata_i_sortiranje AND #Poziv_inicijalizacija AND #Senzor_cilindar_uvučen AND #Senzor_hvataljka_otvorena AND #Home_izvršeno_x AND #Home_izvršeno_y AND (#Trenutna_pozicija_x = 0.0) AND (#Trenutna_pozicija_y = 0.0) THEN
       #Pomicanje_homiranje_x := FALSE;
       #Pomicanje_homiranje_y := FALSE;
       #Zahtjev_za_poziciju := TRUE;
       #Poziv_inicijalizacija := FALSE;
   END_IF;
END_REGION

REGION Network 2: Proces kretnje platforme
   // Zahtjev za dobivanje podataka s Pythona
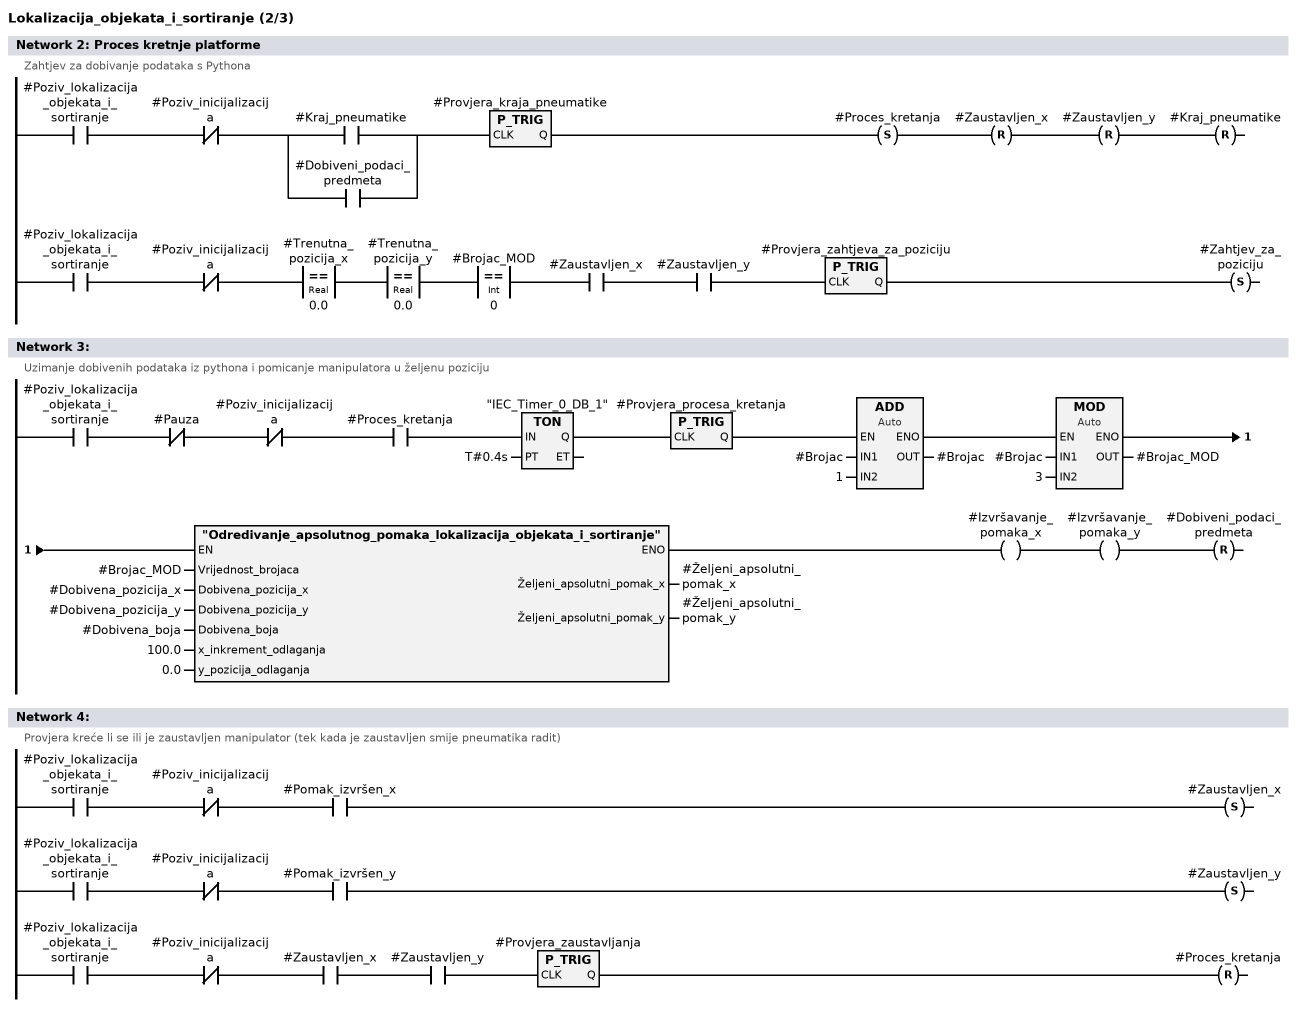
   RUNG wire#powerrail
      Contact( #Poziv_lokalizacija_objekata_i_sortiranje )
      I_Contact( #Poziv_inicijalizacija )
      wire#w1
      Contact( #Kraj_pneumatike )
      wire#w2
      P_Trig( #Provjera_kraja_pneumatike )
      S_Coil( #Proces_kretanja )
      R_Coil( #Zaustavljen_x )
      R_Coil( #Zaustavljen_y )
      R_Coil( #Kraj_pneumatike )
   END_RUNG
   RUNG wire#w1
      Contact( #Dobiveni_podaci_predmeta )
   END_RUNG wire#w2
   RUNG wire#powerrail
      Contact( #Poziv_lokalizacija_objekata_i_sortiranje )
      I_Contact( #Poziv_inicijalizacija )
      { S7_Templates := "SrcType := Real" } EQ_Contact(in1 := #Trenutna_pozicija_x, in2 := 0.0)
      { S7_Templates := "SrcType := Real" } EQ_Contact(in1 := #Trenutna_pozicija_y, in2 := 0.0)
      { S7_Templates := "SrcType := Int" } EQ_Contact(in1 := #Brojac_MOD, in2 := 0)
      Contact( #Zaustavljen_x )
      Contact( #Zaustavljen_y )
      P_Trig( #Provjera_zahtjeva_za_poziciju )
      S_Coil( #Zahtjev_za_poziciju )
   END_RUNG
   // the same network as SCL:
   #_w1 := #Poziv_lokalizacija_objekata_i_sortiranje AND NOT #Poziv_inicijalizacija AND (#Kraj_pneumatike OR #Dobiveni_podaci_predmeta);
   #_w2 := #_w1 AND NOT #Provjera_kraja_pneumatike;   // rising edge
   #Provjera_kraja_pneumatike := #_w1;
   IF #_w2 THEN
       #Proces_kretanja := TRUE;
       #Zaustavljen_x := FALSE;
       #Zaustavljen_y := FALSE;
       #Kraj_pneumatike := FALSE;
   END_IF;
   #_w3 := #Poziv_lokalizacija_objekata_i_sortiranje AND NOT #Poziv_inicijalizacija AND (#Trenutna_pozicija_x = 0.0) AND (#Trenutna_pozicija_y = 0.0) AND (#Brojac_MOD = 0) AND #Zaustavljen_x AND #Zaustavljen_y;
   #_w4 := #_w3 AND NOT #Provjera_zahtjeva_za_poziciju;   // rising edge
   #Provjera_zahtjeva_za_poziciju := #_w3;
   IF #_w4 THEN #Zahtjev_za_poziciju := TRUE; END_IF;
END_REGION

REGION Network 3
   // Uzimanje dobivenih podataka iz pythona i pomicanje manipulatora u željenu poziciju
   "IEC_Timer_0_DB_1".TON(IN := #Poziv_lokalizacija_objekata_i_sortiranje AND NOT #Pauza AND NOT #Poziv_inicijalizacija AND #Proces_kretanja,
                          PT := T#0.4s);
   #_w1 := "IEC_Timer_0_DB_1".Q AND NOT #Provjera_procesa_kretanja;   // rising edge
   #Provjera_procesa_kretanja := "IEC_Timer_0_DB_1".Q;
   IF #_w1 THEN
       #Brojac := #Brojac + 1;
       #Brojac_MOD := #Brojac MOD 3;
   END_IF;
   "Odredivanje_apsolutnog_pomaka_lokalizacija_objekata_i_sortiranje"(EN := #_w1,
                           Vrijednost_brojaca := #Brojac_MOD,
                           Dobivena_pozicija_x := #Dobivena_pozicija_x,
                           Dobivena_pozicija_y := #Dobivena_pozicija_y,
                           Dobivena_boja := #Dobivena_boja,
                           x_inkrement_odlaganja := 100.0,
                           y_pozicija_odlaganja := 0.0,
                           Željeni_apsolutni_pomak_x => #Željeni_apsolutni_pomak_x,
                           Željeni_apsolutni_pomak_y => #Željeni_apsolutni_pomak_y,
                           ENO => #_w2);
   #Izvršavanje_pomaka_x := #_w2;
   #Izvršavanje_pomaka_y := #_w2;
   IF #_w2 THEN #Dobiveni_podaci_predmeta := FALSE; END_IF;
END_REGION

REGION Network 4
   // Provjera kreće li se ili je zaustavljen manipulator (tek kada je zaustavljen smije pneumatika radit)
   RUNG wire#powerrail
      Contact( #Poziv_lokalizacija_objekata_i_sortiranje )
      I_Contact( #Poziv_inicijalizacija )
      Contact( #Pomak_izvršen_x )
      S_Coil( #Zaustavljen_x )
   END_RUNG
   RUNG wire#powerrail
      Contact( #Poziv_lokalizacija_objekata_i_sortiranje )
      I_Contact( #Poziv_inicijalizacija )
      Contact( #Pomak_izvršen_y )
      S_Coil( #Zaustavljen_y )
   END_RUNG
   RUNG wire#powerrail
      Contact( #Poziv_lokalizacija_objekata_i_sortiranje )
      I_Contact( #Poziv_inicijalizacija )
      Contact( #Zaustavljen_x )
      Contact( #Zaustavljen_y )
      P_Trig( #Provjera_zaustavljanja )
      R_Coil( #Proces_kretanja )
   END_RUNG
   // the same network as SCL:
   IF #Poziv_lokalizacija_objekata_i_sortiranje AND NOT #Poziv_inicijalizacija AND #Pomak_izvršen_x THEN
       #Zaustavljen_x := TRUE;
   END_IF;
   IF #Poziv_lokalizacija_objekata_i_sortiranje AND NOT #Poziv_inicijalizacija AND #Pomak_izvršen_y THEN
       #Zaustavljen_y := TRUE;
   END_IF;
   #_w1 := #Poziv_lokalizacija_objekata_i_sortiranje AND NOT #Poziv_inicijalizacija AND #Zaustavljen_x AND #Zaustavljen_y;
   #_w2 := #_w1 AND NOT #Provjera_zaustavljanja;   // rising edge
   #Provjera_zaustavljanja := #_w1;
   IF #_w2 THEN #Proces_kretanja := FALSE; END_IF;
END_REGION

REGION Network 5: Uvjeti aktivacije cilindra i hvataljke tijekom lokalizacije objekata
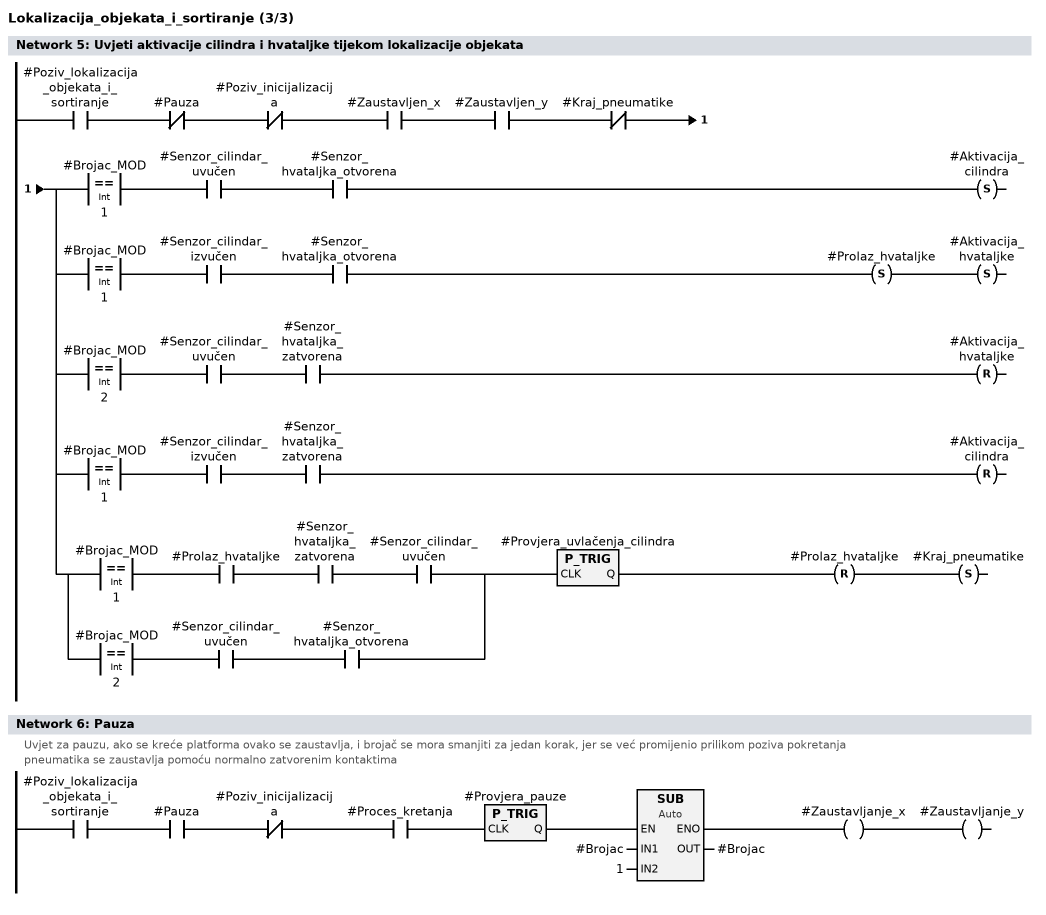
   RUNG wire#powerrail
      Contact( #Poziv_lokalizacija_objekata_i_sortiranje )
      I_Contact( #Pauza )
      I_Contact( #Poziv_inicijalizacija )
      Contact( #Zaustavljen_x )
      Contact( #Zaustavljen_y )
      I_Contact( #Kraj_pneumatike )
      wire#w1
      { S7_Templates := "SrcType := Int" } EQ_Contact(in1 := #Brojac_MOD, in2 := 1)
      Contact( #Senzor_cilindar_uvučen )
      Contact( #Senzor_hvataljka_otvorena )
      S_Coil( #Aktivacija_cilindra )
   END_RUNG
   RUNG wire#w1
      { S7_Templates := "SrcType := Int" } EQ_Contact(in1 := #Brojac_MOD, in2 := 1)
      Contact( #Senzor_cilindar_izvučen )
      Contact( #Senzor_hvataljka_otvorena )
      S_Coil( #Prolaz_hvataljke )
      S_Coil( #Aktivacija_hvataljke )
   END_RUNG
   RUNG wire#w1
      { S7_Templates := "SrcType := Int" } EQ_Contact(in1 := #Brojac_MOD, in2 := 2)
      Contact( #Senzor_cilindar_uvučen )
      Contact( #Senzor_hvataljka_zatvorena )
      R_Coil( #Aktivacija_hvataljke )
   END_RUNG
   RUNG wire#w1
      { S7_Templates := "SrcType := Int" } EQ_Contact(in1 := #Brojac_MOD, in2 := 1)
      Contact( #Senzor_cilindar_izvučen )
      Contact( #Senzor_hvataljka_zatvorena )
      R_Coil( #Aktivacija_cilindra )
   END_RUNG
   RUNG wire#w1
      { S7_Templates := "SrcType := Int" } EQ_Contact(in1 := #Brojac_MOD, in2 := 1)
      Contact( #Prolaz_hvataljke )
      Contact( #Senzor_hvataljka_zatvorena )
      Contact( #Senzor_cilindar_uvučen )
      wire#w2
      P_Trig( #Provjera_uvlačenja_cilindra )
      R_Coil( #Prolaz_hvataljke )
      S_Coil( #Kraj_pneumatike )
   END_RUNG
   RUNG wire#w1
      { S7_Templates := "SrcType := Int" } EQ_Contact(in1 := #Brojac_MOD, in2 := 2)
      Contact( #Senzor_cilindar_uvučen )
      Contact( #Senzor_hvataljka_otvorena )
   END_RUNG wire#w2
   // the same network as SCL:
   #_w1 := #Poziv_lokalizacija_objekata_i_sortiranje AND NOT #Pauza AND NOT #Poziv_inicijalizacija AND #Zaustavljen_x AND #Zaustavljen_y AND NOT #Kraj_pneumatike;
   IF #_w1 AND (#Brojac_MOD = 1) AND #Senzor_cilindar_uvučen AND #Senzor_hvataljka_otvorena THEN
       #Aktivacija_cilindra := TRUE;
   END_IF;
   IF #_w1 AND (#Brojac_MOD = 1) AND #Senzor_cilindar_izvučen AND #Senzor_hvataljka_otvorena THEN
       #Prolaz_hvataljke := TRUE;
       #Aktivacija_hvataljke := TRUE;
   END_IF;
   IF #_w1 AND (#Brojac_MOD = 2) AND #Senzor_cilindar_uvučen AND #Senzor_hvataljka_zatvorena THEN
       #Aktivacija_hvataljke := FALSE;
   END_IF;
   IF #_w1 AND (#Brojac_MOD = 1) AND #Senzor_cilindar_izvučen AND #Senzor_hvataljka_zatvorena THEN
       #Aktivacija_cilindra := FALSE;
   END_IF;
   #_w2 := #_w1 AND (((#Brojac_MOD = 1) AND #Prolaz_hvataljke AND #Senzor_hvataljka_zatvorena AND #Senzor_cilindar_uvučen) OR ((#Brojac_MOD = 2) AND #Senzor_cilindar_uvučen AND #Senzor_hvataljka_otvorena));
   #_w3 := #_w2 AND NOT #Provjera_uvlačenja_cilindra;   // rising edge
   #Provjera_uvlačenja_cilindra := #_w2;
   IF #_w3 THEN
       #Prolaz_hvataljke := FALSE;
       #Kraj_pneumatike := TRUE;
   END_IF;
END_REGION

REGION Network 6: Pauza
   // Uvjet za pauzu, ako se kreće platforma ovako se zaustavlja, i brojač se mora smanjiti za jedan korak, jer se već promijenio prilikom poziva pokretanja
   // pneumatika se zaustavlja pomoću normalno zatvorenim kontaktima
   RUNG wire#powerrail
      Contact( #Poziv_lokalizacija_objekata_i_sortiranje )
      Contact( #Pauza )
      I_Contact( #Poziv_inicijalizacija )
      Contact( #Proces_kretanja )
      P_Trig( #Provjera_pauze )
      Sub(in1 := #Brojac, in2 := 1, out => #Brojac)
      Coil( #Zaustavljanje_x )
      Coil( #Zaustavljanje_y )
   END_RUNG
   // the same network as SCL:
   #_w1 := #Poziv_lokalizacija_objekata_i_sortiranje AND #Pauza AND NOT #Poziv_inicijalizacija AND #Proces_kretanja;
   #_w2 := #_w1 AND NOT #Provjera_pauze;   // rising edge
   #Provjera_pauze := #_w1;
   IF #_w2 THEN #Brojac := #Brojac - 1; END_IF;
   #Zaustavljanje_x := #_w2;
   #Zaustavljanje_y := #_w2;
END_REGION
END_FUNCTION_BLOCK

FUNCTION_BLOCK "Paletizacija"   // FB5, LAD
{ S7_Optimized_Access := 'TRUE' }
VERSION : 0.1
   VAR_INPUT
      Senzor_cilindar_uvučen : Bool;
      Senzor_cilindar_izvučen : Bool;
      Senzor_hvataljka_zatvorena : Bool;
      Senzor_hvataljka_otvorena : Bool;
      Home_izvršeno_x : Bool;
      Home_izvršeno_y : Bool;
      Trenutna_pozicija_x : Real;
      Trenutna_pozicija_y : Real;
      Pomak_izvršen_x : Bool;
      Pomak_izvršen_y : Bool;
      Broj_komada_palete_x : Int;   // 1...6
      Broj_komada_palete_y : Int;   // 1...3
      Koordinata_palete_izuzimanja_x : Real;   // Vrijednost x koordinate izuzimanja
      Koordinata_palete_izuzimanja_y : Real;   // Vrijednost y koordinate izuzimanja
      Koordinata_palete_odlaganja_x : Real;   // Vrijednost x koordinate odlaganja za prvi predmet
      Koordinata_palete_odlaganja_y : Real;   // Vrijednost y koordinate odlaganja za prvi predmet
      Pauza : Bool;
   END_VAR
   VAR_OUTPUT
      Aktivacija_cilindra : Bool;   // 1 - izvučen, 0 - uvučen
      Aktivacija_hvataljke : Bool;   // 1 - zatvorena, 0 - otvorena
      Home_x : Bool;
      Home_y : Bool;
      Željeni_apsolutni_pomak_x : Real;
      Željeni_apsolutni_pomak_y : Real;
      Izvršavanje_pomaka_x : Bool;
      Izvršavanje_pomaka_y : Bool;
      Zaustavljanje_x : Bool;
      Zaustavljanje_y : Bool;
      Kraj_paletizacije : Bool;
   END_VAR
   VAR_IN_OUT
      Poziv_paletizacija : Bool;
   END_VAR
   VAR
      Poziv_inicijalizacija : Bool;
      brojac : Int := 0;
      Provjera_parnosti : Int;   // 0 je paran, 1 je neparan
      Provjera_poziva_paletizacije : Bool;
      Provjera_starta_paletizacije : Bool;
      Provjera_kraja_pneumatike : Bool;
      Provjera_uvlačenja_cilindra : Bool;
      Proces_kretanja : Bool;
      Provjera_procesa_kretanja : Bool;
      Zaustavljen_x : Bool;
      Zaustavljen_y : Bool;
      Kraj_pneumatike : Bool;
      Zadnji_korak : Int;   // 2N+1
      Prolaz_cilindra : Bool := 0;
      Prolaz_hvataljke : Bool := 0;   // Provjera je li hvataljka bila aktivirana tijekom koraka pneumatike, bez ove varijable bila bi dva identična pozivanja pa se nebi znalo ima li hvataljka uhvaćen predmet ili ne
      Provjera_zaustavljanja : Bool;
   END_VAR
   VAR_TEMP
      Pomicanje_homiranje_x : Bool;
      Pomicanje_homiranje_y : Bool;
      Cilindar_je_uvucen : Bool;
      Hvataljka_je_otvorena : Bool;
   END_VAR
   VAR CONSTANT
      Udaljenost_po_x : Real := 35.0;   // određuje koliko predmeti mogu biti udaljeni međusobno po x osi
      Udaljenost_po_y : Real := 70.0;   // određuje koliko predmeti mogu biti udaljeni međusobno po y osi
   END_VAR
   VAR_TEMP   // added for the SCL form of the ladder/FBD networks
      _w1 : Bool;
      _w2 : Bool;
      _w3 : Bool;
      _w4 : Bool;
   END_VAR
BEGIN

REGION Network 1: Pokretanje paletizacije i inicijalizacija
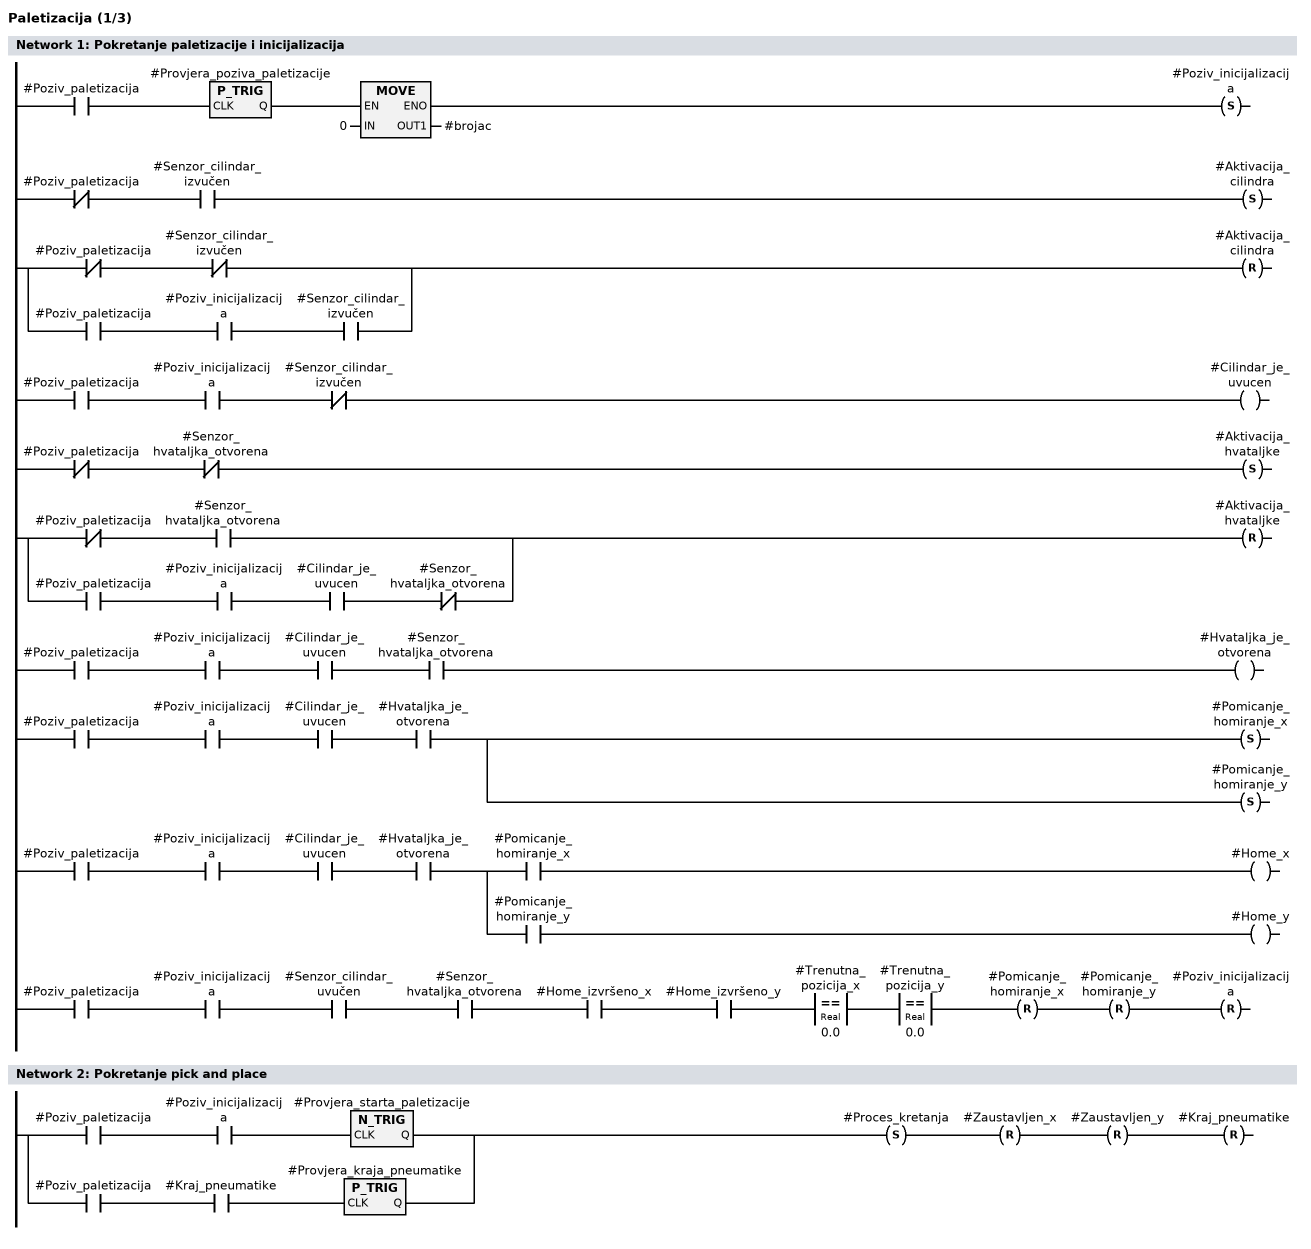
   RUNG wire#powerrail
      Contact( #Poziv_paletizacija )
      P_Trig( #Provjera_poziva_paletizacije )
      Move(in := 0, out1 => #brojac)
      S_Coil( #Poziv_inicijalizacija )
   END_RUNG
   RUNG wire#powerrail
      I_Contact( #Poziv_paletizacija )
      Contact( #Senzor_cilindar_izvučen )
      S_Coil( #Aktivacija_cilindra )
   END_RUNG
   RUNG wire#powerrail
      I_Contact( #Poziv_paletizacija )
      I_Contact( #Senzor_cilindar_izvučen )
      wire#w1
      R_Coil( #Aktivacija_cilindra )
   END_RUNG
   RUNG wire#powerrail
      Contact( #Poziv_paletizacija )
      Contact( #Poziv_inicijalizacija )
      Contact( #Senzor_cilindar_izvučen )
   END_RUNG wire#w1
   RUNG wire#powerrail
      Contact( #Poziv_paletizacija )
      Contact( #Poziv_inicijalizacija )
      I_Contact( #Senzor_cilindar_izvučen )
      Coil( #Cilindar_je_uvucen )
   END_RUNG
   RUNG wire#powerrail
      I_Contact( #Poziv_paletizacija )
      I_Contact( #Senzor_hvataljka_otvorena )
      S_Coil( #Aktivacija_hvataljke )
   END_RUNG
   RUNG wire#powerrail
      I_Contact( #Poziv_paletizacija )
      Contact( #Senzor_hvataljka_otvorena )
      wire#w2
      R_Coil( #Aktivacija_hvataljke )
   END_RUNG
   RUNG wire#powerrail
      Contact( #Poziv_paletizacija )
      Contact( #Poziv_inicijalizacija )
      Contact( #Cilindar_je_uvucen )
      I_Contact( #Senzor_hvataljka_otvorena )
   END_RUNG wire#w2
   RUNG wire#powerrail
      Contact( #Poziv_paletizacija )
      Contact( #Poziv_inicijalizacija )
      Contact( #Cilindar_je_uvucen )
      Contact( #Senzor_hvataljka_otvorena )
      Coil( #Hvataljka_je_otvorena )
   END_RUNG
   RUNG wire#powerrail
      Contact( #Poziv_paletizacija )
      Contact( #Poziv_inicijalizacija )
      Contact( #Cilindar_je_uvucen )
      Contact( #Hvataljka_je_otvorena )
      wire#w3
      S_Coil( #Pomicanje_homiranje_x )
   END_RUNG
   RUNG wire#w3
      S_Coil( #Pomicanje_homiranje_y )
   END_RUNG
   RUNG wire#powerrail
      Contact( #Poziv_paletizacija )
      Contact( #Poziv_inicijalizacija )
      Contact( #Cilindar_je_uvucen )
      Contact( #Hvataljka_je_otvorena )
      wire#w4
      Contact( #Pomicanje_homiranje_x )
      Coil( #Home_x )
   END_RUNG
   RUNG wire#w4
      Contact( #Pomicanje_homiranje_y )
      Coil( #Home_y )
   END_RUNG
   RUNG wire#powerrail
      Contact( #Poziv_paletizacija )
      Contact( #Poziv_inicijalizacija )
      Contact( #Senzor_cilindar_uvučen )
      Contact( #Senzor_hvataljka_otvorena )
      Contact( #Home_izvršeno_x )
      Contact( #Home_izvršeno_y )
      { S7_Templates := "SrcType := Real" } EQ_Contact(in1 := #Trenutna_pozicija_x, in2 := 0.0)
      { S7_Templates := "SrcType := Real" } EQ_Contact(in1 := #Trenutna_pozicija_y, in2 := 0.0)
      R_Coil( #Pomicanje_homiranje_x )
      R_Coil( #Pomicanje_homiranje_y )
      R_Coil( #Poziv_inicijalizacija )
   END_RUNG
   // the same network as SCL:
   #_w1 := #Poziv_paletizacija AND NOT #Provjera_poziva_paletizacije;   // rising edge
   #Provjera_poziva_paletizacije := #Poziv_paletizacija;
   IF #_w1 THEN
       #brojac := 0;
       #Poziv_inicijalizacija := TRUE;
   END_IF;
   IF NOT #Poziv_paletizacija AND #Senzor_cilindar_izvučen THEN #Aktivacija_cilindra := TRUE; END_IF;
   IF (NOT #Poziv_paletizacija AND NOT #Senzor_cilindar_izvučen) OR (#Poziv_paletizacija AND #Poziv_inicijalizacija AND #Senzor_cilindar_izvučen) THEN
       #Aktivacija_cilindra := FALSE;
   END_IF;
   #Cilindar_je_uvucen := #Poziv_paletizacija AND #Poziv_inicijalizacija AND NOT #Senzor_cilindar_izvučen;
   IF NOT #Poziv_paletizacija AND NOT #Senzor_hvataljka_otvorena THEN #Aktivacija_hvataljke := TRUE; END_IF;
   IF (NOT #Poziv_paletizacija AND #Senzor_hvataljka_otvorena) OR (#Poziv_paletizacija AND #Poziv_inicijalizacija AND #Cilindar_je_uvucen AND NOT #Senzor_hvataljka_otvorena) THEN
       #Aktivacija_hvataljke := FALSE;
   END_IF;
   #Hvataljka_je_otvorena := #Poziv_paletizacija AND #Poziv_inicijalizacija AND #Cilindar_je_uvucen AND #Senzor_hvataljka_otvorena;
   IF #Poziv_paletizacija AND #Poziv_inicijalizacija AND #Cilindar_je_uvucen AND #Hvataljka_je_otvorena THEN
       #Pomicanje_homiranje_x := TRUE;
       #Pomicanje_homiranje_y := TRUE;
   END_IF;
   #_w2 := #Poziv_paletizacija AND #Poziv_inicijalizacija AND #Cilindar_je_uvucen AND #Hvataljka_je_otvorena;
   #Home_x := #_w2 AND #Pomicanje_homiranje_x;
   #Home_y := #_w2 AND #Pomicanje_homiranje_y;
   IF #Poziv_paletizacija AND #Poziv_inicijalizacija AND #Senzor_cilindar_uvučen AND #Senzor_hvataljka_otvorena AND #Home_izvršeno_x AND #Home_izvršeno_y AND (#Trenutna_pozicija_x = 0.0) AND (#Trenutna_pozicija_y = 0.0) THEN
       #Pomicanje_homiranje_x := FALSE;
       #Pomicanje_homiranje_y := FALSE;
       #Poziv_inicijalizacija := FALSE;
   END_IF;
END_REGION

REGION Network 2: Pokretanje pick and place
   RUNG wire#powerrail
      Contact( #Poziv_paletizacija )
      Contact( #Poziv_inicijalizacija )
      N_Trig( #Provjera_starta_paletizacije )
      wire#w1
      S_Coil( #Proces_kretanja )
      R_Coil( #Zaustavljen_x )
      R_Coil( #Zaustavljen_y )
      R_Coil( #Kraj_pneumatike )
   END_RUNG
   RUNG wire#powerrail
      Contact( #Poziv_paletizacija )
      Contact( #Kraj_pneumatike )
      P_Trig( #Provjera_kraja_pneumatike )
   END_RUNG wire#w1
   // the same network as SCL:
   #_w1 := #Poziv_paletizacija AND #Poziv_inicijalizacija;
   #_w2 := NOT #_w1 AND #Provjera_starta_paletizacije;   // falling edge
   #Provjera_starta_paletizacije := #_w1;
   #_w3 := #Poziv_paletizacija AND #Kraj_pneumatike;
   #_w4 := #_w3 AND NOT #Provjera_kraja_pneumatike;   // rising edge
   #Provjera_kraja_pneumatike := #_w3;
   IF #_w2 OR #_w4 THEN
       #Proces_kretanja := TRUE;
       #Zaustavljen_x := FALSE;
       #Zaustavljen_y := FALSE;
       #Kraj_pneumatike := FALSE;
   END_IF;
END_REGION

REGION Network 3
   // Funkcija s dijeljenjem; određuje os koja će se prva ispunjavat (ako y gledamo kao ulaz, onda se x redak ispunjava, a ako se gleda x kao ulaz, onda se y stupac ispunjava)
   // Funkcija s mod; određuje os koja će ispunjavati pozicije unutar prvog reda ili stupca
   // VAŽNO!! u obje funkcije treba postaviti isti broj komada palete za odlaganje da bi ispravno radilo
   // npr. 12 komada; paleta (x=4, y=3) s ulazom od broja x u paleti (4): mod=012301230123, div=000011112222, a brojke na istoj poziciji su koordinate koje se povecaju za 1: (1,1), (2,1), (3,1)...,(4,3)
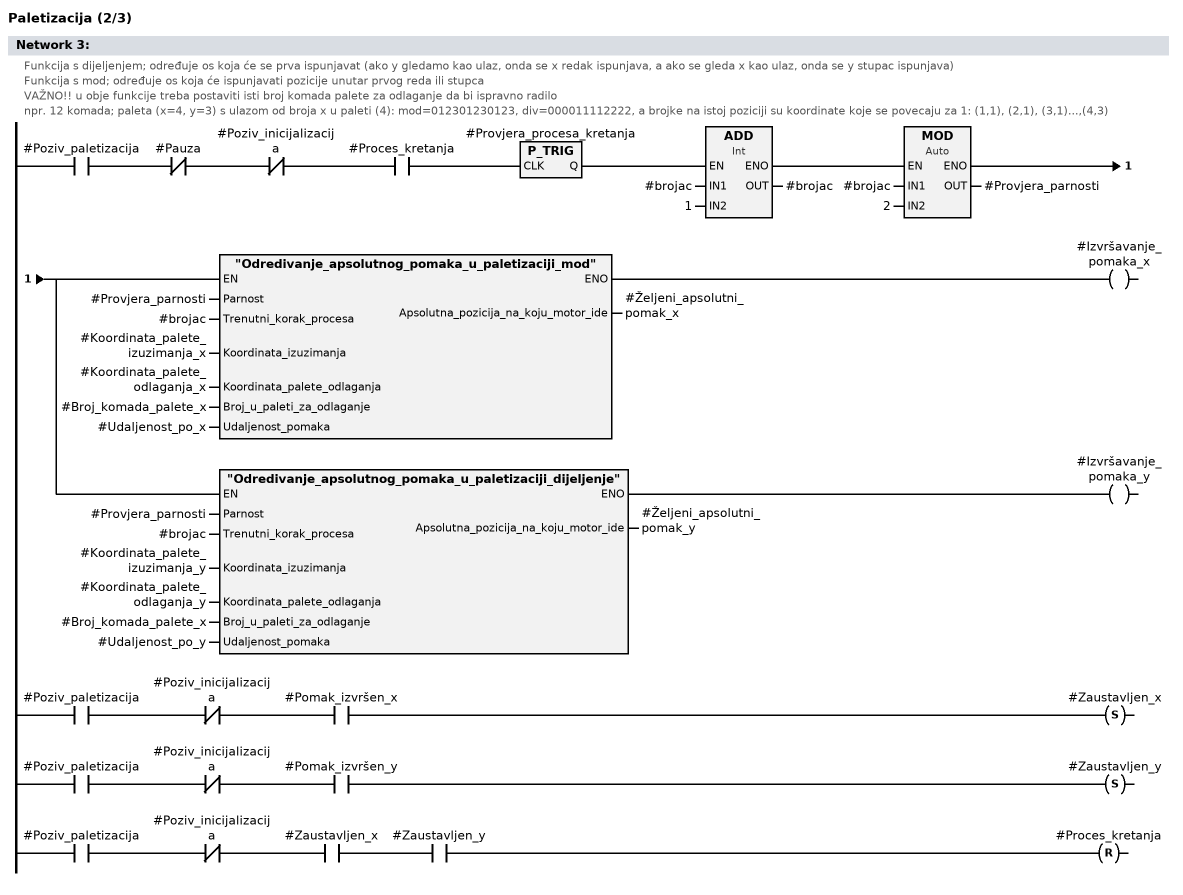
   RUNG wire#powerrail
      Contact( #Poziv_paletizacija )
      I_Contact( #Pauza )
      I_Contact( #Poziv_inicijalizacija )
      Contact( #Proces_kretanja )
      P_Trig( #Provjera_procesa_kretanja )
      { S7_Templates := "SrcType := Int" } Add(in1 := #brojac, in2 := 1, out => #brojac)
      Mod(in1 := #brojac, in2 := 2, out => #Provjera_parnosti)
      wire#w1
      "Odredivanje_apsolutnog_pomaka_u_paletizaciji_mod"(Parnost := #Provjera_parnosti, Trenutni_korak_procesa := #brojac, Koordinata_izuzimanja := #Koordinata_palete_izuzimanja_x, Koordinata_palete_odlaganja := #Koordinata_palete_odlaganja_x, Broj_u_paleti_za_odlaganje := #Broj_komada_palete_x, Udaljenost_pomaka := #Udaljenost_po_x, Apsolutna_pozicija_na_koju_motor_ide => #Željeni_apsolutni_pomak_x)
      Coil( #Izvršavanje_pomaka_x )
   END_RUNG
   RUNG wire#w1
      "Odredivanje_apsolutnog_pomaka_u_paletizaciji_dijeljenje"(Parnost := #Provjera_parnosti, Trenutni_korak_procesa := #brojac, Koordinata_izuzimanja := #Koordinata_palete_izuzimanja_y, Koordinata_palete_odlaganja := #Koordinata_palete_odlaganja_y, Broj_u_paleti_za_odlaganje := #Broj_komada_palete_x, Udaljenost_pomaka := #Udaljenost_po_y, Apsolutna_pozicija_na_koju_motor_ide => #Željeni_apsolutni_pomak_y)
      Coil( #Izvršavanje_pomaka_y )
   END_RUNG
   RUNG wire#powerrail
      Contact( #Poziv_paletizacija )
      I_Contact( #Poziv_inicijalizacija )
      Contact( #Pomak_izvršen_x )
      S_Coil( #Zaustavljen_x )
   END_RUNG
   RUNG wire#powerrail
      Contact( #Poziv_paletizacija )
      I_Contact( #Poziv_inicijalizacija )
      Contact( #Pomak_izvršen_y )
      S_Coil( #Zaustavljen_y )
   END_RUNG
   RUNG wire#powerrail
      Contact( #Poziv_paletizacija )
      I_Contact( #Poziv_inicijalizacija )
      Contact( #Zaustavljen_x )
      Contact( #Zaustavljen_y )
      R_Coil( #Proces_kretanja )
   END_RUNG
   // the same network as SCL:
   #_w1 := #Poziv_paletizacija AND NOT #Pauza AND NOT #Poziv_inicijalizacija AND #Proces_kretanja;
   #_w2 := #_w1 AND NOT #Provjera_procesa_kretanja;   // rising edge
   #Provjera_procesa_kretanja := #_w1;
   IF #_w2 THEN
       #brojac := #brojac + 1;
       #Provjera_parnosti := #brojac MOD 2;
   END_IF;
   "Odredivanje_apsolutnog_pomaka_u_paletizaciji_mod"(EN := #_w2,
                           Parnost := #Provjera_parnosti,
                           Trenutni_korak_procesa := #brojac,
                           Koordinata_izuzimanja := #Koordinata_palete_izuzimanja_x,
                           Koordinata_palete_odlaganja := #Koordinata_palete_odlaganja_x,
                           Broj_u_paleti_za_odlaganje := #Broj_komada_palete_x,
                           Udaljenost_pomaka := #Udaljenost_po_x,
                           Apsolutna_pozicija_na_koju_motor_ide => #Željeni_apsolutni_pomak_x,
                           ENO => #_w3);
   #Izvršavanje_pomaka_x := #_w3;
   "Odredivanje_apsolutnog_pomaka_u_paletizaciji_dijeljenje"(EN := #_w2,
                           Parnost := #Provjera_parnosti,
                           Trenutni_korak_procesa := #brojac,
                           Koordinata_izuzimanja := #Koordinata_palete_izuzimanja_y,
                           Koordinata_palete_odlaganja := #Koordinata_palete_odlaganja_y,
                           Broj_u_paleti_za_odlaganje := #Broj_komada_palete_x,
                           Udaljenost_pomaka := #Udaljenost_po_y,
                           Apsolutna_pozicija_na_koju_motor_ide => #Željeni_apsolutni_pomak_y,
                           ENO => #_w4);
   #Izvršavanje_pomaka_y := #_w4;
   IF #Poziv_paletizacija AND NOT #Poziv_inicijalizacija AND #Pomak_izvršen_x THEN
       #Zaustavljen_x := TRUE;
   END_IF;
   IF #Poziv_paletizacija AND NOT #Poziv_inicijalizacija AND #Pomak_izvršen_y THEN
       #Zaustavljen_y := TRUE;
   END_IF;
   IF #Poziv_paletizacija AND NOT #Poziv_inicijalizacija AND #Zaustavljen_x AND #Zaustavljen_y THEN
       #Proces_kretanja := FALSE;
   END_IF;
END_REGION

REGION Network 4: Uvjeti aktivacije cilindra i hvataljke tijekom paletizacije
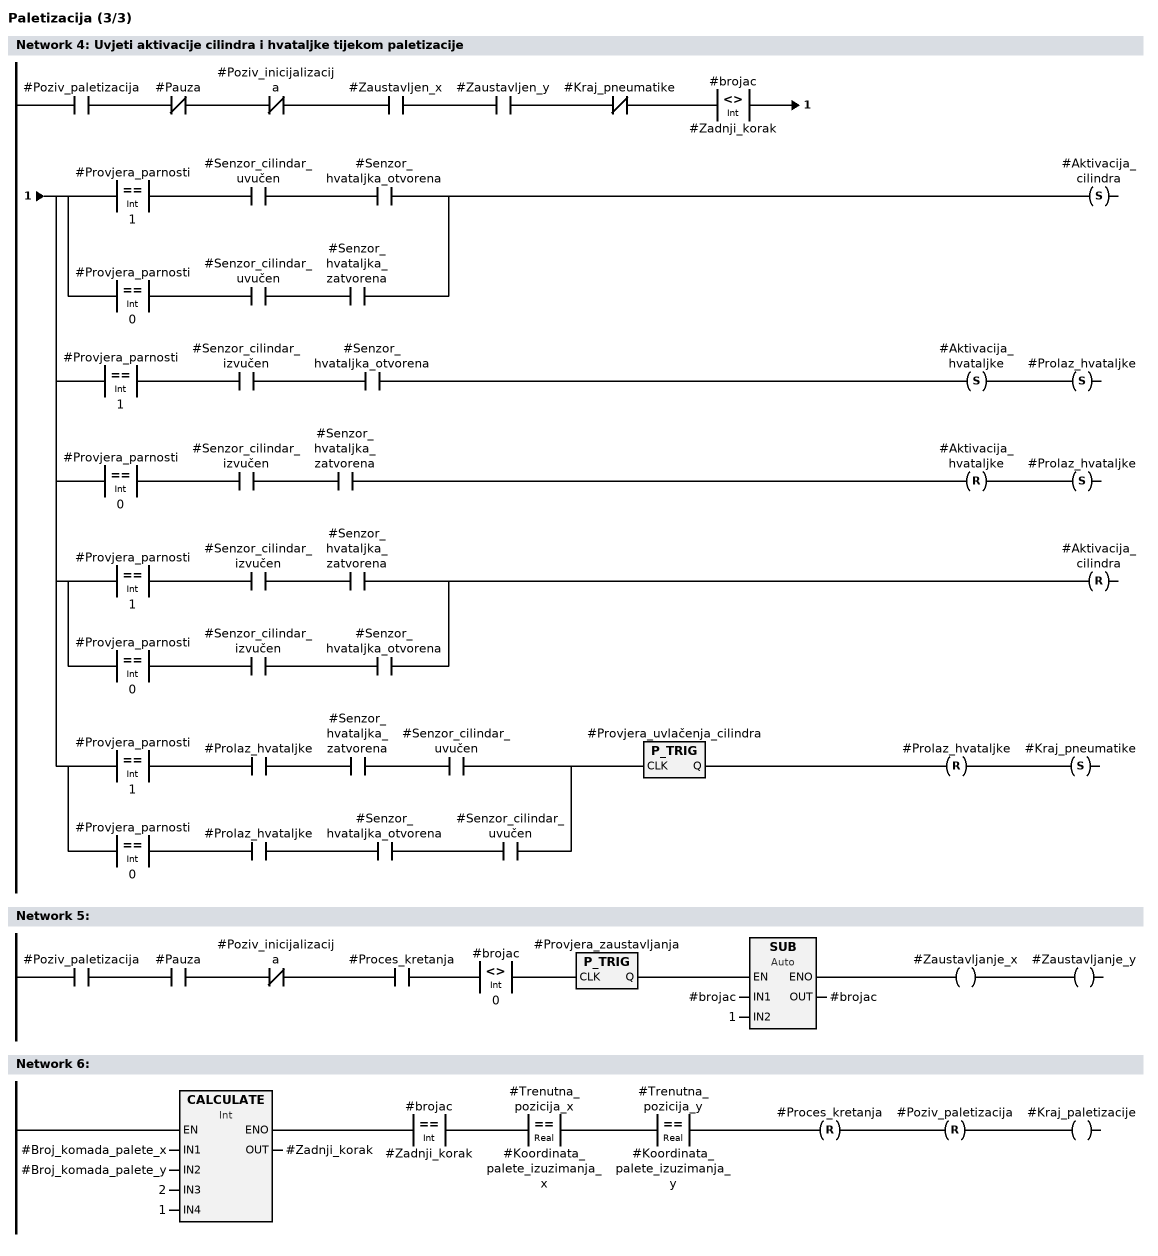
   RUNG wire#powerrail
      Contact( #Poziv_paletizacija )
      I_Contact( #Pauza )
      I_Contact( #Poziv_inicijalizacija )
      Contact( #Zaustavljen_x )
      Contact( #Zaustavljen_y )
      I_Contact( #Kraj_pneumatike )
      { S7_Templates := "SrcType := Int" } NE_Contact(in1 := #brojac, in2 := #Zadnji_korak)
      wire#w1
      { S7_Templates := "SrcType := Int" } EQ_Contact(in1 := #Provjera_parnosti, in2 := 1)
      Contact( #Senzor_cilindar_uvučen )
      Contact( #Senzor_hvataljka_otvorena )
      wire#w2
      S_Coil( #Aktivacija_cilindra )
   END_RUNG
   RUNG wire#w1
      { S7_Templates := "SrcType := Int" } EQ_Contact(in1 := #Provjera_parnosti, in2 := 0)
      Contact( #Senzor_cilindar_uvučen )
      Contact( #Senzor_hvataljka_zatvorena )
   END_RUNG wire#w2
   RUNG wire#w1
      { S7_Templates := "SrcType := Int" } EQ_Contact(in1 := #Provjera_parnosti, in2 := 1)
      Contact( #Senzor_cilindar_izvučen )
      Contact( #Senzor_hvataljka_otvorena )
      S_Coil( #Aktivacija_hvataljke )
      S_Coil( #Prolaz_hvataljke )
   END_RUNG
   RUNG wire#w1
      { S7_Templates := "SrcType := Int" } EQ_Contact(in1 := #Provjera_parnosti, in2 := 0)
      Contact( #Senzor_cilindar_izvučen )
      Contact( #Senzor_hvataljka_zatvorena )
      R_Coil( #Aktivacija_hvataljke )
      S_Coil( #Prolaz_hvataljke )
   END_RUNG
   RUNG wire#w1
      { S7_Templates := "SrcType := Int" } EQ_Contact(in1 := #Provjera_parnosti, in2 := 1)
      Contact( #Senzor_cilindar_izvučen )
      Contact( #Senzor_hvataljka_zatvorena )
      wire#w3
      R_Coil( #Aktivacija_cilindra )
   END_RUNG
   RUNG wire#w1
      { S7_Templates := "SrcType := Int" } EQ_Contact(in1 := #Provjera_parnosti, in2 := 0)
      Contact( #Senzor_cilindar_izvučen )
      Contact( #Senzor_hvataljka_otvorena )
   END_RUNG wire#w3
   RUNG wire#w1
      { S7_Templates := "SrcType := Int" } EQ_Contact(in1 := #Provjera_parnosti, in2 := 1)
      Contact( #Prolaz_hvataljke )
      Contact( #Senzor_hvataljka_zatvorena )
      Contact( #Senzor_cilindar_uvučen )
      wire#w4
      P_Trig( #Provjera_uvlačenja_cilindra )
      R_Coil( #Prolaz_hvataljke )
      S_Coil( #Kraj_pneumatike )
   END_RUNG
   RUNG wire#w1
      { S7_Templates := "SrcType := Int" } EQ_Contact(in1 := #Provjera_parnosti, in2 := 0)
      Contact( #Prolaz_hvataljke )
      Contact( #Senzor_hvataljka_otvorena )
      Contact( #Senzor_cilindar_uvučen )
   END_RUNG wire#w4
   // the same network as SCL:
   #_w1 := #Poziv_paletizacija AND NOT #Pauza AND NOT #Poziv_inicijalizacija AND #Zaustavljen_x AND #Zaustavljen_y AND NOT #Kraj_pneumatike AND (#brojac <> #Zadnji_korak);
   IF #_w1 AND (((#Provjera_parnosti = 1) AND #Senzor_cilindar_uvučen AND #Senzor_hvataljka_otvorena) OR ((#Provjera_parnosti = 0) AND #Senzor_cilindar_uvučen AND #Senzor_hvataljka_zatvorena)) THEN
       #Aktivacija_cilindra := TRUE;
   END_IF;
   IF #_w1 AND (#Provjera_parnosti = 1) AND #Senzor_cilindar_izvučen AND #Senzor_hvataljka_otvorena THEN
       #Aktivacija_hvataljke := TRUE;
       #Prolaz_hvataljke := TRUE;
   END_IF;
   IF #_w1 AND (#Provjera_parnosti = 0) AND #Senzor_cilindar_izvučen AND #Senzor_hvataljka_zatvorena THEN
       #Aktivacija_hvataljke := FALSE;
       #Prolaz_hvataljke := TRUE;
   END_IF;
   IF #_w1 AND (((#Provjera_parnosti = 1) AND #Senzor_cilindar_izvučen AND #Senzor_hvataljka_zatvorena) OR ((#Provjera_parnosti = 0) AND #Senzor_cilindar_izvučen AND #Senzor_hvataljka_otvorena)) THEN
       #Aktivacija_cilindra := FALSE;
   END_IF;
   #_w2 := #_w1 AND (((#Provjera_parnosti = 1) AND #Prolaz_hvataljke AND #Senzor_hvataljka_zatvorena AND #Senzor_cilindar_uvučen) OR ((#Provjera_parnosti = 0) AND #Prolaz_hvataljke AND #Senzor_hvataljka_otvorena AND #Senzor_cilindar_uvučen));
   #_w3 := #_w2 AND NOT #Provjera_uvlačenja_cilindra;   // rising edge
   #Provjera_uvlačenja_cilindra := #_w2;
   IF #_w3 THEN
       #Prolaz_hvataljke := FALSE;
       #Kraj_pneumatike := TRUE;
   END_IF;
END_REGION

REGION Network 5
   RUNG wire#powerrail
      Contact( #Poziv_paletizacija )
      Contact( #Pauza )
      I_Contact( #Poziv_inicijalizacija )
      Contact( #Proces_kretanja )
      { S7_Templates := "SrcType := Int" } NE_Contact(in1 := #brojac, in2 := 0)
      P_Trig( #Provjera_zaustavljanja )
      Sub(in1 := #brojac, in2 := 1, out => #brojac)
      Coil( #Zaustavljanje_x )
      Coil( #Zaustavljanje_y )
   END_RUNG
   // the same network as SCL:
   #_w1 := #Poziv_paletizacija AND #Pauza AND NOT #Poziv_inicijalizacija AND #Proces_kretanja AND (#brojac <> 0);
   #_w2 := #_w1 AND NOT #Provjera_zaustavljanja;   // rising edge
   #Provjera_zaustavljanja := #_w1;
   IF #_w2 THEN #brojac := #brojac - 1; END_IF;
   #Zaustavljanje_x := #_w2;
   #Zaustavljanje_y := #_w2;
END_REGION

REGION Network 6
   RUNG wire#powerrail
      { S7_Templates := "SrcType := Int"; S7_Expression := "IN1*IN2*IN3+IN4" } Calculate(in1 := #Broj_komada_palete_x, in2 := #Broj_komada_palete_y, in3 := 2, in4 := 1, out => #Zadnji_korak)
      { S7_Templates := "SrcType := Int" } EQ_Contact(in1 := #brojac, in2 := #Zadnji_korak)
      { S7_Templates := "SrcType := Real" } EQ_Contact(in1 := #Trenutna_pozicija_x, in2 := #Koordinata_palete_izuzimanja_x)
      { S7_Templates := "SrcType := Real" } EQ_Contact(in1 := #Trenutna_pozicija_y, in2 := #Koordinata_palete_izuzimanja_y)
      R_Coil( #Proces_kretanja )
      R_Coil( #Poziv_paletizacija )
      Coil( #Kraj_paletizacije )
   END_RUNG
   // the same network as SCL:
   #Zadnji_korak := #Broj_komada_palete_x*#Broj_komada_palete_y*2+1;
   #_w1 := (#brojac = #Zadnji_korak) AND (#Trenutna_pozicija_x = #Koordinata_palete_izuzimanja_x) AND (#Trenutna_pozicija_y = #Koordinata_palete_izuzimanja_y);
   IF #_w1 THEN
       #Proces_kretanja := FALSE;
       #Poziv_paletizacija := FALSE;
   END_IF;
   #Kraj_paletizacije := #_w1;
END_REGION
END_FUNCTION_BLOCK

FUNCTION "Odredivanje_apsolutnog_pomaka_u_paletizaciji_dijeljenje" : Void   // FC1, LAD
{ S7_Optimized_Access := 'TRUE' }
VERSION : 0.1
// Paletizacija je podijeljena na dva koraka pomicanja, mjesto izuzimanja i mjesto odlaganja predmeta - logika opisana u FB bloku Paletizacija
   VAR_INPUT
      Parnost : Int;   // 0 je paran, 1 je neparan
      Trenutni_korak_procesa : Int;   // [1, 2N+1] gdje je N broj komada za plaetizaciju
      Koordinata_izuzimanja : Real;
      Koordinata_palete_odlaganja : Real;
      Broj_u_paleti_za_odlaganje : Int;   // za x 1...6; za y 1...3 - to je broj s kojim se modira
      Udaljenost_pomaka : Real;   // 35 ili 65 ovisno o x ili y osi
   END_VAR
   VAR_OUTPUT
      Apsolutna_pozicija_na_koju_motor_ide : Real;
   END_VAR
   VAR_TEMP
      Dijeljenje : Int;
      Korak_u_odlaganju : Int;
   END_VAR
BEGIN

REGION Network 1
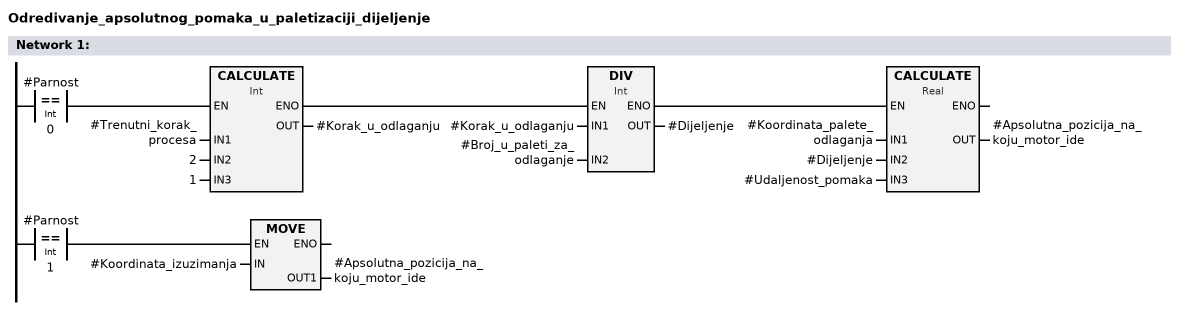
   RUNG wire#powerrail
      { S7_Templates := "SrcType := Int" } EQ_Contact(in1 := #Parnost, in2 := 0)
      { S7_Templates := "SrcType := Int"; S7_Expression := "IN1/IN2-IN3" } Calculate(in1 := #Trenutni_korak_procesa, in2 := 2, in3 := 1, out => #Korak_u_odlaganju)
      { S7_Templates := "SrcType := Int" } Div(in1 := #Korak_u_odlaganju, in2 := #Broj_u_paleti_za_odlaganje, out => #Dijeljenje)
      { S7_Templates := "SrcType := Real"; S7_Expression := "IN1+IN2*IN3" } Calculate(in1 := #Koordinata_palete_odlaganja, in2 := #Dijeljenje, in3 := #Udaljenost_pomaka, out => #Apsolutna_pozicija_na_koju_motor_ide)
   END_RUNG
   RUNG wire#powerrail
      { S7_Templates := "SrcType := Int" } EQ_Contact(in1 := #Parnost, in2 := 1)
      Move(in := #Koordinata_izuzimanja, out1 => #Apsolutna_pozicija_na_koju_motor_ide)
   END_RUNG
   // the same network as SCL:
   IF #Parnost = 0 THEN
       #Korak_u_odlaganju := #Trenutni_korak_procesa/2-1;
       #Dijeljenje := #Korak_u_odlaganju / #Broj_u_paleti_za_odlaganje;
       #Apsolutna_pozicija_na_koju_motor_ide := #Koordinata_palete_odlaganja+#Dijeljenje*#Udaljenost_pomaka;
   END_IF;
   IF #Parnost = 1 THEN #Apsolutna_pozicija_na_koju_motor_ide := #Koordinata_izuzimanja; END_IF;
END_REGION
END_FUNCTION

FUNCTION "Pneumatski_cilindar_upravljanje" : Void   // FC2, LAD
{ S7_Optimized_Access := 'TRUE' }
VERSION : 0.1
   VAR_INPUT
      Zahtjev_uvlačenje_cilindra : Bool;
      Zahtjev_izvlačenje_cilindra : Bool;
      Senzor_izvučeni_cilindar : Bool;
      Senzor_uvučeni_cilindar : Bool;
   END_VAR
   VAR_OUTPUT
      Izvlačenje_cilindra : Bool;
      Uvlačenje_cilindra : Bool;
   END_VAR
   VAR_TEMP
      Akcija_izvlačenja : Bool;
      Akcija_uvlačenja : Bool;
   END_VAR
BEGIN

REGION Network 1
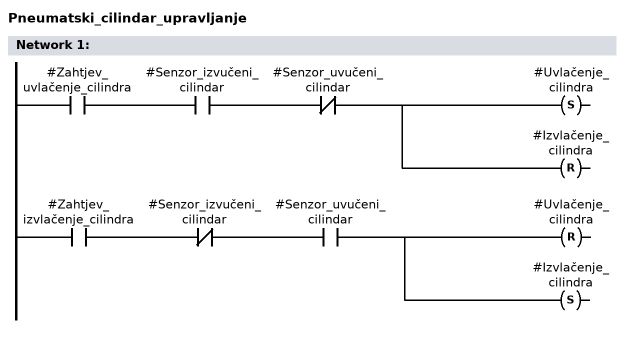
   RUNG wire#powerrail
      Contact( #Zahtjev_uvlačenje_cilindra )
      Contact( #Senzor_izvučeni_cilindar )
      I_Contact( #Senzor_uvučeni_cilindar )
      wire#w1
      S_Coil( #Uvlačenje_cilindra )
   END_RUNG
   RUNG wire#w1
      R_Coil( #Izvlačenje_cilindra )
   END_RUNG
   RUNG wire#powerrail
      Contact( #Zahtjev_izvlačenje_cilindra )
      I_Contact( #Senzor_izvučeni_cilindar )
      Contact( #Senzor_uvučeni_cilindar )
      wire#w2
      R_Coil( #Uvlačenje_cilindra )
   END_RUNG
   RUNG wire#w2
      S_Coil( #Izvlačenje_cilindra )
   END_RUNG
   // the same network as SCL:
   IF #Zahtjev_uvlačenje_cilindra AND #Senzor_izvučeni_cilindar AND NOT #Senzor_uvučeni_cilindar THEN
       #Uvlačenje_cilindra := TRUE;
       #Izvlačenje_cilindra := FALSE;
   END_IF;
   IF #Zahtjev_izvlačenje_cilindra AND NOT #Senzor_izvučeni_cilindar AND #Senzor_uvučeni_cilindar THEN
       #Uvlačenje_cilindra := FALSE;
       #Izvlačenje_cilindra := TRUE;
   END_IF;
END_REGION
END_FUNCTION

FUNCTION "Hvataljka_upravljanje" : Void   // FC3, LAD
{ S7_Optimized_Access := 'TRUE' }
VERSION : 0.1
   VAR_INPUT
      Zahtjev_otvaranje_hvataljke : Bool;
      Zahtjev_zatvaranje_hvataljke : Bool;
      Senzor_zatvorena_hvataljka : Bool;
      Senzor_otvorena_hvataljka : Bool;
   END_VAR
   VAR_OUTPUT
      Zatvaranje_hvataljke : Bool;
      Otvaranje_hvataljke : Bool;
   END_VAR
BEGIN

REGION Network 1
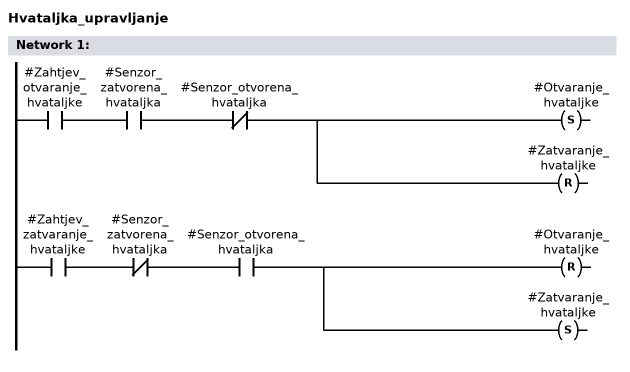
   RUNG wire#powerrail
      Contact( #Zahtjev_otvaranje_hvataljke )
      Contact( #Senzor_zatvorena_hvataljka )
      I_Contact( #Senzor_otvorena_hvataljka )
      wire#w1
      S_Coil( #Otvaranje_hvataljke )
   END_RUNG
   RUNG wire#w1
      R_Coil( #Zatvaranje_hvataljke )
   END_RUNG
   RUNG wire#powerrail
      Contact( #Zahtjev_zatvaranje_hvataljke )
      I_Contact( #Senzor_zatvorena_hvataljka )
      Contact( #Senzor_otvorena_hvataljka )
      wire#w2
      R_Coil( #Otvaranje_hvataljke )
   END_RUNG
   RUNG wire#w2
      S_Coil( #Zatvaranje_hvataljke )
   END_RUNG
   // the same network as SCL:
   IF #Zahtjev_otvaranje_hvataljke AND #Senzor_zatvorena_hvataljka AND NOT #Senzor_otvorena_hvataljka THEN
       #Otvaranje_hvataljke := TRUE;
       #Zatvaranje_hvataljke := FALSE;
   END_IF;
   IF #Zahtjev_zatvaranje_hvataljke AND NOT #Senzor_zatvorena_hvataljka AND #Senzor_otvorena_hvataljka THEN
       #Otvaranje_hvataljke := FALSE;
       #Zatvaranje_hvataljke := TRUE;
   END_IF;
END_REGION
END_FUNCTION

FUNCTION "Odredivanje_apsolutnog_pomaka_u_paletizaciji_mod" : Void   // FC4, LAD
{ S7_Optimized_Access := 'TRUE' }
VERSION : 0.1
// Paletizacija je podijeljena na dva koraka pomicanja, mjesto izuzimanja i mjesto odlaganja predmeta - logika opisana u FB bloku Paletizacija
   VAR_INPUT
      Parnost : Int;   // 0 je paran, 1 je neparan
      Trenutni_korak_procesa : Int;   // [1, 2N+1] gdje je N broj komada za plaetizaciju
      Koordinata_izuzimanja : Real;
      Koordinata_palete_odlaganja : Real;
      Broj_u_paleti_za_odlaganje : Int;   // za x 1...6; za y 1...3 - to je broj s kojim se modira
      Udaljenost_pomaka : Real;   // 35 ili 65 ovisno o x ili y osi
   END_VAR
   VAR_OUTPUT
      Apsolutna_pozicija_na_koju_motor_ide : Real;
   END_VAR
   VAR_TEMP
      "Mod" : Int;
      Korak_u_odlaganju : Int;
   END_VAR
BEGIN

REGION Network 1
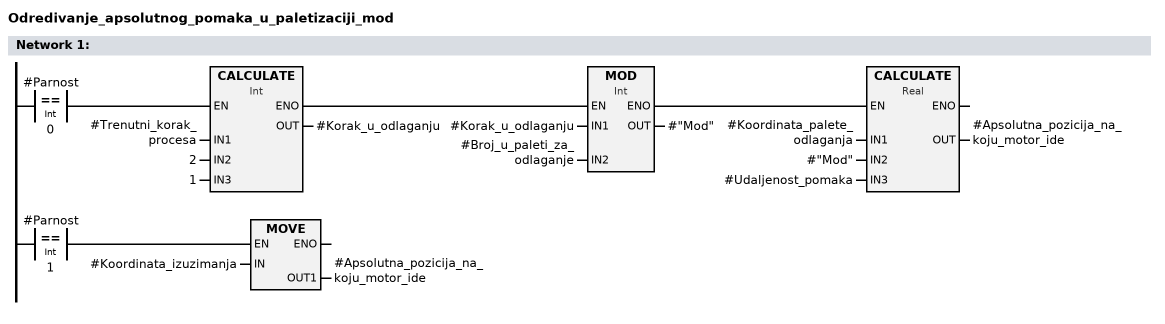
   RUNG wire#powerrail
      { S7_Templates := "SrcType := Int" } EQ_Contact(in1 := #Parnost, in2 := 0)
      { S7_Templates := "SrcType := Int"; S7_Expression := "IN1/IN2-IN3" } Calculate(in1 := #Trenutni_korak_procesa, in2 := 2, in3 := 1, out => #Korak_u_odlaganju)
      { S7_Templates := "SrcType := Int" } Mod(in1 := #Korak_u_odlaganju, in2 := #Broj_u_paleti_za_odlaganje, out => #"Mod")
      { S7_Templates := "SrcType := Real"; S7_Expression := "IN1+IN2*IN3" } Calculate(in1 := #Koordinata_palete_odlaganja, in2 := #"Mod", in3 := #Udaljenost_pomaka, out => #Apsolutna_pozicija_na_koju_motor_ide)
   END_RUNG
   RUNG wire#powerrail
      { S7_Templates := "SrcType := Int" } EQ_Contact(in1 := #Parnost, in2 := 1)
      Move(in := #Koordinata_izuzimanja, out1 => #Apsolutna_pozicija_na_koju_motor_ide)
   END_RUNG
   // the same network as SCL:
   IF #Parnost = 0 THEN
       #Korak_u_odlaganju := #Trenutni_korak_procesa/2-1;
       #"Mod" := #Korak_u_odlaganju MOD #Broj_u_paleti_za_odlaganje;
       #Apsolutna_pozicija_na_koju_motor_ide := #Koordinata_palete_odlaganja+#"Mod"*#Udaljenost_pomaka;
   END_IF;
   IF #Parnost = 1 THEN #Apsolutna_pozicija_na_koju_motor_ide := #Koordinata_izuzimanja; END_IF;
END_REGION
END_FUNCTION

FUNCTION "Odredivanje_apsolutnog_pomaka_lokalizacija_objekata_i_sortiranje" : Void   // FC5, LAD
{ S7_Optimized_Access := 'TRUE' }
VERSION : 0.1
// Lokalizacija objekata je podijeljena u tri koraka pomicanja: nula, mjesto uzimanja predmeta i mjesto odlaganja predmeta
   VAR_INPUT
      Vrijednost_brojaca : Int;
      Dobivena_pozicija_x : Real;
      Dobivena_pozicija_y : Real;
      Dobivena_boja : Int;
      x_inkrement_odlaganja : Real;
      y_pozicija_odlaganja : Real;
   END_VAR
   VAR_OUTPUT
      Željeni_apsolutni_pomak_x : Real;
      Željeni_apsolutni_pomak_y : Real;
   END_VAR
BEGIN

REGION Network 1
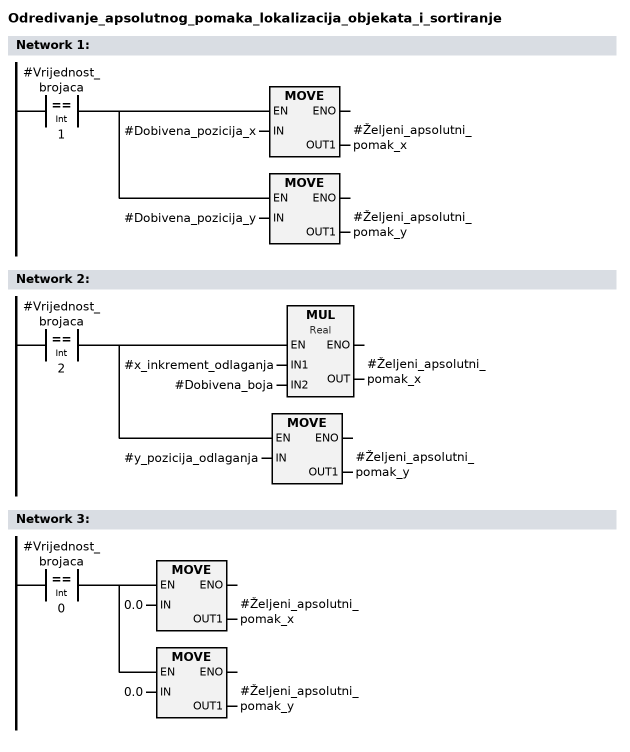
   RUNG wire#powerrail
      { S7_Templates := "SrcType := Int" } EQ_Contact(in1 := #Vrijednost_brojaca, in2 := 1)
      wire#w1
      Move(in := #Dobivena_pozicija_x, out1 => #Željeni_apsolutni_pomak_x)
   END_RUNG
   RUNG wire#w1
      Move(in := #Dobivena_pozicija_y, out1 => #Željeni_apsolutni_pomak_y)
   END_RUNG
   // the same network as SCL:
   IF #Vrijednost_brojaca = 1 THEN
       #Željeni_apsolutni_pomak_x := #Dobivena_pozicija_x;
       #Željeni_apsolutni_pomak_y := #Dobivena_pozicija_y;
   END_IF;
END_REGION

REGION Network 2
   RUNG wire#powerrail
      { S7_Templates := "SrcType := Int" } EQ_Contact(in1 := #Vrijednost_brojaca, in2 := 2)
      wire#w1
      { S7_Templates := "SrcType := Real" } Mul(in1 := #x_inkrement_odlaganja, in2 := #Dobivena_boja, out => #Željeni_apsolutni_pomak_x)
   END_RUNG
   RUNG wire#w1
      Move(in := #y_pozicija_odlaganja, out1 => #Željeni_apsolutni_pomak_y)
   END_RUNG
   // the same network as SCL:
   IF #Vrijednost_brojaca = 2 THEN
       #Željeni_apsolutni_pomak_x := #x_inkrement_odlaganja * #Dobivena_boja;
       #Željeni_apsolutni_pomak_y := #y_pozicija_odlaganja;
   END_IF;
END_REGION

REGION Network 3
   RUNG wire#powerrail
      { S7_Templates := "SrcType := Int" } EQ_Contact(in1 := #Vrijednost_brojaca, in2 := 0)
      wire#w1
      Move(in := 0.0, out1 => #Željeni_apsolutni_pomak_x)
   END_RUNG
   RUNG wire#w1
      Move(in := 0.0, out1 => #Željeni_apsolutni_pomak_y)
   END_RUNG
   // the same network as SCL:
   IF #Vrijednost_brojaca = 0 THEN
       #Željeni_apsolutni_pomak_x := 0.0;
       #Željeni_apsolutni_pomak_y := 0.0;
   END_IF;
END_REGION
END_FUNCTION

ORGANIZATION_BLOCK "Main"   // OB1, LAD, ProgramCycle
TITLE = "Main Program Sweep (Cycle)"
{ S7_Optimized_Access := 'TRUE' }
VERSION : 0.1
   VAR_INPUT
      Initial_Call : Bool;   // Initial call of this OB
      Remanence : Bool;   // =True, if remanent data are available
   END_VAR
   VAR_TEMP   // added for the SCL form of the ladder/FBD networks
      _w1 : Bool;
      _w2 : Bool;
      _w3 : Bool;
      _w4 : Bool;
      _w5 : Bool;
   END_VAR
BEGIN

REGION Network 1: Motor upravljanje x osi
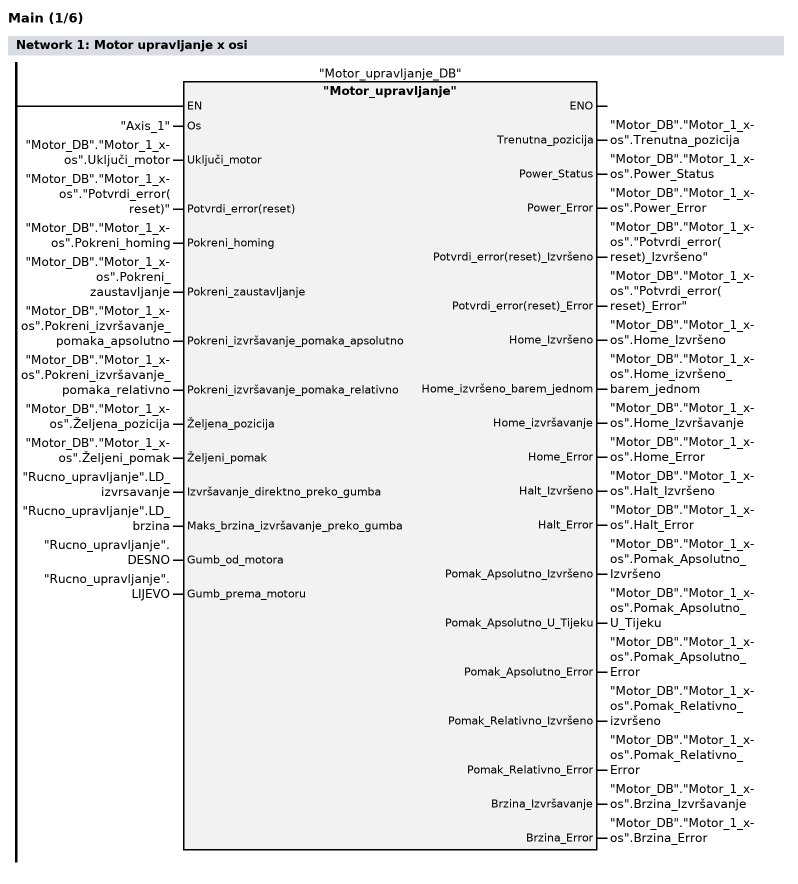
   RUNG wire#powerrail
      "Motor_upravljanje_DB"(Os := "Axis_1", Uključi_motor := "Motor_DB"."Motor_1_x-os".Uključi_motor, "Potvrdi_error(reset)" := "Motor_DB"."Motor_1_x-os"."Potvrdi_error(reset)", Pokreni_homing := "Motor_DB"."Motor_1_x-os".Pokreni_homing, Pokreni_zaustavljanje := "Motor_DB"."Motor_1_x-os".Pokreni_zaustavljanje, Pokreni_izvršavanje_pomaka_apsolutno := "Motor_DB"."Motor_1_x-os".Pokreni_izvršavanje_pomaka_apsolutno, Pokreni_izvršavanje_pomaka_relativno := "Motor_DB"."Motor_1_x-os".Pokreni_izvršavanje_pomaka_relativno, Željena_pozicija := "Motor_DB"."Motor_1_x-os".Željena_pozicija, Željeni_pomak := "Motor_DB"."Motor_1_x-os".Željeni_pomak, Izvršavanje_direktno_preko_gumba := "Rucno_upravljanje".LD_izvrsavanje, Maks_brzina_izvršavanje_preko_gumba := "Rucno_upravljanje".LD_brzina, Gumb_od_motora := "Rucno_upravljanje".DESNO, Gumb_prema_motoru := "Rucno_upravljanje".LIJEVO, Trenutna_pozicija => "Motor_DB"."Motor_1_x-os".Trenutna_pozicija, Power_Status => "Motor_DB"."Motor_1_x-os".Power_Status, Power_Error => "Motor_DB"."Motor_1_x-os".Power_Error, "Potvrdi_error(reset)_Izvršeno" => "Motor_DB"."Motor_1_x-os"."Potvrdi_error(reset)_Izvršeno", "Potvrdi_error(reset)_Error" => "Motor_DB"."Motor_1_x-os"."Potvrdi_error(reset)_Error", Home_Izvršeno => "Motor_DB"."Motor_1_x-os".Home_Izvršeno, Home_izvršeno_barem_jednom => "Motor_DB"."Motor_1_x-os".Home_izvršeno_barem_jednom, Home_izvršavanje => "Motor_DB"."Motor_1_x-os".Home_Izvršavanje, Home_Error => "Motor_DB"."Motor_1_x-os".Home_Error, Halt_Izvršeno => "Motor_DB"."Motor_1_x-os".Halt_Izvršeno, Halt_Error => "Motor_DB"."Motor_1_x-os".Halt_Error, Pomak_Apsolutno_Izvršeno => "Motor_DB"."Motor_1_x-os".Pomak_Apsolutno_Izvršeno, Pomak_Apsolutno_U_Tijeku => "Motor_DB"."Motor_1_x-os".Pomak_Apsolutno_U_Tijeku, Pomak_Apsolutno_Error => "Motor_DB"."Motor_1_x-os".Pomak_Apsolutno_Error, Pomak_Relativno_Izvršeno => "Motor_DB"."Motor_1_x-os".Pomak_Relativno_izvršeno, Pomak_Relativno_Error => "Motor_DB"."Motor_1_x-os".Pomak_Relativno_Error, Brzina_Izvršavanje => "Motor_DB"."Motor_1_x-os".Brzina_Izvršavanje, Brzina_Error => "Motor_DB"."Motor_1_x-os".Brzina_Error)
   END_RUNG
   // the same network as SCL:
   "Motor_upravljanje_DB"(Os := "Axis_1",   // "Motor_upravljanje"
                          Uključi_motor := "Motor_DB"."Motor_1_x-os".Uključi_motor,
                          "Potvrdi_error(reset)" := "Motor_DB"."Motor_1_x-os"."Potvrdi_error(reset)",
                          Pokreni_homing := "Motor_DB"."Motor_1_x-os".Pokreni_homing,
                          Pokreni_zaustavljanje := "Motor_DB"."Motor_1_x-os".Pokreni_zaustavljanje,
                          Pokreni_izvršavanje_pomaka_apsolutno := "Motor_DB"."Motor_1_x-os".Pokreni_izvršavanje_pomaka_apsolutno,
                          Pokreni_izvršavanje_pomaka_relativno := "Motor_DB"."Motor_1_x-os".Pokreni_izvršavanje_pomaka_relativno,
                          Željena_pozicija := "Motor_DB"."Motor_1_x-os".Željena_pozicija,
                          Željeni_pomak := "Motor_DB"."Motor_1_x-os".Željeni_pomak,
                          Izvršavanje_direktno_preko_gumba := "Rucno_upravljanje".LD_izvrsavanje,
                          Maks_brzina_izvršavanje_preko_gumba := "Rucno_upravljanje".LD_brzina,
                          Gumb_od_motora := "Rucno_upravljanje".DESNO,
                          Gumb_prema_motoru := "Rucno_upravljanje".LIJEVO,
                          Trenutna_pozicija => "Motor_DB"."Motor_1_x-os".Trenutna_pozicija,
                          Power_Status => "Motor_DB"."Motor_1_x-os".Power_Status,
                          Power_Error => "Motor_DB"."Motor_1_x-os".Power_Error,
                          "Potvrdi_error(reset)_Izvršeno" => "Motor_DB"."Motor_1_x-os"."Potvrdi_error(reset)_Izvršeno",
                          "Potvrdi_error(reset)_Error" => "Motor_DB"."Motor_1_x-os"."Potvrdi_error(reset)_Error",
                          Home_Izvršeno => "Motor_DB"."Motor_1_x-os".Home_Izvršeno,
                          Home_izvršeno_barem_jednom => "Motor_DB"."Motor_1_x-os".Home_izvršeno_barem_jednom,
                          Home_izvršavanje => "Motor_DB"."Motor_1_x-os".Home_Izvršavanje,
                          Home_Error => "Motor_DB"."Motor_1_x-os".Home_Error,
                          Halt_Izvršeno => "Motor_DB"."Motor_1_x-os".Halt_Izvršeno,
                          Halt_Error => "Motor_DB"."Motor_1_x-os".Halt_Error,
                          Pomak_Apsolutno_Izvršeno => "Motor_DB"."Motor_1_x-os".Pomak_Apsolutno_Izvršeno,
                          Pomak_Apsolutno_U_Tijeku => "Motor_DB"."Motor_1_x-os".Pomak_Apsolutno_U_Tijeku,
                          Pomak_Apsolutno_Error => "Motor_DB"."Motor_1_x-os".Pomak_Apsolutno_Error,
                          Pomak_Relativno_Izvršeno => "Motor_DB"."Motor_1_x-os".Pomak_Relativno_izvršeno,
                          Pomak_Relativno_Error => "Motor_DB"."Motor_1_x-os".Pomak_Relativno_Error,
                          Brzina_Izvršavanje => "Motor_DB"."Motor_1_x-os".Brzina_Izvršavanje,
                          Brzina_Error => "Motor_DB"."Motor_1_x-os".Brzina_Error);
END_REGION

REGION Network 2: Motor upravljanje y osi
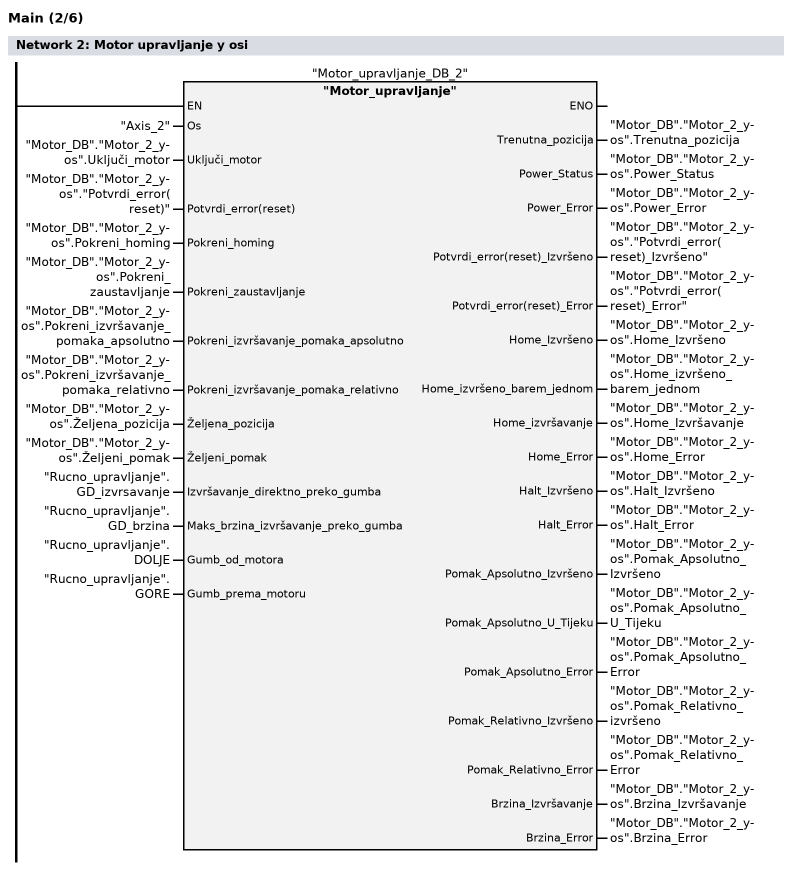
   RUNG wire#powerrail
      "Motor_upravljanje_DB_2"(Os := "Axis_2", Uključi_motor := "Motor_DB"."Motor_2_y-os".Uključi_motor, "Potvrdi_error(reset)" := "Motor_DB"."Motor_2_y-os"."Potvrdi_error(reset)", Pokreni_homing := "Motor_DB"."Motor_2_y-os".Pokreni_homing, Pokreni_zaustavljanje := "Motor_DB"."Motor_2_y-os".Pokreni_zaustavljanje, Pokreni_izvršavanje_pomaka_apsolutno := "Motor_DB"."Motor_2_y-os".Pokreni_izvršavanje_pomaka_apsolutno, Pokreni_izvršavanje_pomaka_relativno := "Motor_DB"."Motor_2_y-os".Pokreni_izvršavanje_pomaka_relativno, Željena_pozicija := "Motor_DB"."Motor_2_y-os".Željena_pozicija, Željeni_pomak := "Motor_DB"."Motor_2_y-os".Željeni_pomak, Izvršavanje_direktno_preko_gumba := "Rucno_upravljanje".GD_izvrsavanje, Maks_brzina_izvršavanje_preko_gumba := "Rucno_upravljanje".GD_brzina, Gumb_od_motora := "Rucno_upravljanje".DOLJE, Gumb_prema_motoru := "Rucno_upravljanje".GORE, Trenutna_pozicija => "Motor_DB"."Motor_2_y-os".Trenutna_pozicija, Power_Status => "Motor_DB"."Motor_2_y-os".Power_Status, Power_Error => "Motor_DB"."Motor_2_y-os".Power_Error, "Potvrdi_error(reset)_Izvršeno" => "Motor_DB"."Motor_2_y-os"."Potvrdi_error(reset)_Izvršeno", "Potvrdi_error(reset)_Error" => "Motor_DB"."Motor_2_y-os"."Potvrdi_error(reset)_Error", Home_Izvršeno => "Motor_DB"."Motor_2_y-os".Home_Izvršeno, Home_izvršeno_barem_jednom => "Motor_DB"."Motor_2_y-os".Home_izvršeno_barem_jednom, Home_izvršavanje => "Motor_DB"."Motor_2_y-os".Home_Izvršavanje, Home_Error => "Motor_DB"."Motor_2_y-os".Home_Error, Halt_Izvršeno => "Motor_DB"."Motor_2_y-os".Halt_Izvršeno, Halt_Error => "Motor_DB"."Motor_2_y-os".Halt_Error, Pomak_Apsolutno_Izvršeno => "Motor_DB"."Motor_2_y-os".Pomak_Apsolutno_Izvršeno, Pomak_Apsolutno_U_Tijeku => "Motor_DB"."Motor_2_y-os".Pomak_Apsolutno_U_Tijeku, Pomak_Apsolutno_Error => "Motor_DB"."Motor_2_y-os".Pomak_Apsolutno_Error, Pomak_Relativno_Izvršeno => "Motor_DB"."Motor_2_y-os".Pomak_Relativno_izvršeno, Pomak_Relativno_Error => "Motor_DB"."Motor_2_y-os".Pomak_Relativno_Error, Brzina_Izvršavanje => "Motor_DB"."Motor_2_y-os".Brzina_Izvršavanje, Brzina_Error => "Motor_DB"."Motor_2_y-os".Brzina_Error)
   END_RUNG
   // the same network as SCL:
   "Motor_upravljanje_DB_2"(Os := "Axis_2",   // "Motor_upravljanje"
                           Uključi_motor := "Motor_DB"."Motor_2_y-os".Uključi_motor,
                           "Potvrdi_error(reset)" := "Motor_DB"."Motor_2_y-os"."Potvrdi_error(reset)",
                           Pokreni_homing := "Motor_DB"."Motor_2_y-os".Pokreni_homing,
                           Pokreni_zaustavljanje := "Motor_DB"."Motor_2_y-os".Pokreni_zaustavljanje,
                           Pokreni_izvršavanje_pomaka_apsolutno := "Motor_DB"."Motor_2_y-os".Pokreni_izvršavanje_pomaka_apsolutno,
                           Pokreni_izvršavanje_pomaka_relativno := "Motor_DB"."Motor_2_y-os".Pokreni_izvršavanje_pomaka_relativno,
                           Željena_pozicija := "Motor_DB"."Motor_2_y-os".Željena_pozicija,
                           Željeni_pomak := "Motor_DB"."Motor_2_y-os".Željeni_pomak,
                           Izvršavanje_direktno_preko_gumba := "Rucno_upravljanje".GD_izvrsavanje,
                           Maks_brzina_izvršavanje_preko_gumba := "Rucno_upravljanje".GD_brzina,
                           Gumb_od_motora := "Rucno_upravljanje".DOLJE,
                           Gumb_prema_motoru := "Rucno_upravljanje".GORE,
                           Trenutna_pozicija => "Motor_DB"."Motor_2_y-os".Trenutna_pozicija,
                           Power_Status => "Motor_DB"."Motor_2_y-os".Power_Status,
                           Power_Error => "Motor_DB"."Motor_2_y-os".Power_Error,
                           "Potvrdi_error(reset)_Izvršeno" => "Motor_DB"."Motor_2_y-os"."Potvrdi_error(reset)_Izvršeno",
                           "Potvrdi_error(reset)_Error" => "Motor_DB"."Motor_2_y-os"."Potvrdi_error(reset)_Error",
                           Home_Izvršeno => "Motor_DB"."Motor_2_y-os".Home_Izvršeno,
                           Home_izvršeno_barem_jednom => "Motor_DB"."Motor_2_y-os".Home_izvršeno_barem_jednom,
                           Home_izvršavanje => "Motor_DB"."Motor_2_y-os".Home_Izvršavanje,
                           Home_Error => "Motor_DB"."Motor_2_y-os".Home_Error,
                           Halt_Izvršeno => "Motor_DB"."Motor_2_y-os".Halt_Izvršeno,
                           Halt_Error => "Motor_DB"."Motor_2_y-os".Halt_Error,
                           Pomak_Apsolutno_Izvršeno => "Motor_DB"."Motor_2_y-os".Pomak_Apsolutno_Izvršeno,
                           Pomak_Apsolutno_U_Tijeku => "Motor_DB"."Motor_2_y-os".Pomak_Apsolutno_U_Tijeku,
                           Pomak_Apsolutno_Error => "Motor_DB"."Motor_2_y-os".Pomak_Apsolutno_Error,
                           Pomak_Relativno_Izvršeno => "Motor_DB"."Motor_2_y-os".Pomak_Relativno_izvršeno,
                           Pomak_Relativno_Error => "Motor_DB"."Motor_2_y-os".Pomak_Relativno_Error,
                           Brzina_Izvršavanje => "Motor_DB"."Motor_2_y-os".Brzina_Izvršavanje,
                           Brzina_Error => "Motor_DB"."Motor_2_y-os".Brzina_Error);
END_REGION

REGION Network 3: Paletizacija
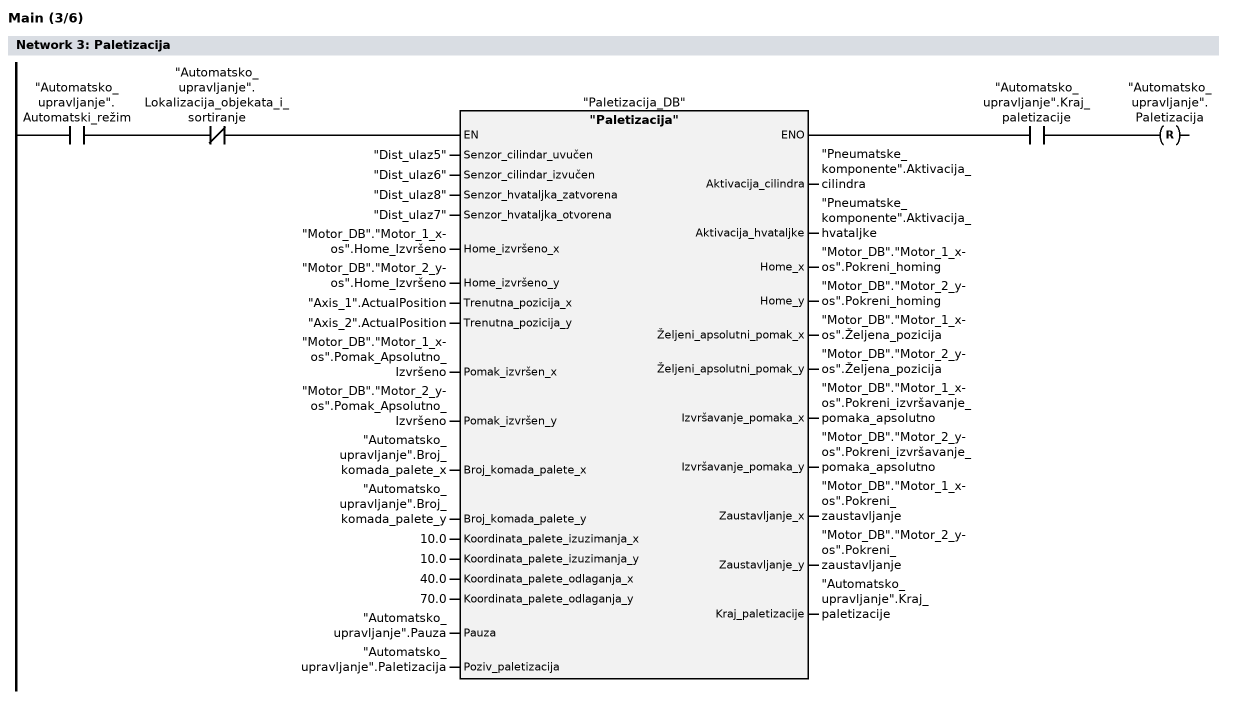
   RUNG wire#powerrail
      Contact( "Automatsko_upravljanje".Automatski_režim )
      I_Contact( "Automatsko_upravljanje".Lokalizacija_objekata_i_sortiranje )
      "Paletizacija_DB"(Senzor_cilindar_uvučen := "Dist_ulaz5", Senzor_cilindar_izvučen := "Dist_ulaz6", Senzor_hvataljka_zatvorena := "Dist_ulaz8", Senzor_hvataljka_otvorena := "Dist_ulaz7", Home_izvršeno_x := "Motor_DB"."Motor_1_x-os".Home_Izvršeno, Home_izvršeno_y := "Motor_DB"."Motor_2_y-os".Home_Izvršeno, Trenutna_pozicija_x := "Axis_1".ActualPosition, Trenutna_pozicija_y := "Axis_2".ActualPosition, Pomak_izvršen_x := "Motor_DB"."Motor_1_x-os".Pomak_Apsolutno_Izvršeno, Pomak_izvršen_y := "Motor_DB"."Motor_2_y-os".Pomak_Apsolutno_Izvršeno, Broj_komada_palete_x := "Automatsko_upravljanje".Broj_komada_palete_x, Broj_komada_palete_y := "Automatsko_upravljanje".Broj_komada_palete_y, Koordinata_palete_izuzimanja_x := 10.0, Koordinata_palete_izuzimanja_y := 10.0, Koordinata_palete_odlaganja_x := 40.0, Koordinata_palete_odlaganja_y := 70.0, Pauza := "Automatsko_upravljanje".Pauza, Poziv_paletizacija := "Automatsko_upravljanje".Paletizacija, Aktivacija_cilindra => "Pneumatske_komponente".Aktivacija_cilindra, Aktivacija_hvataljke => "Pneumatske_komponente".Aktivacija_hvataljke, Home_x => "Motor_DB"."Motor_1_x-os".Pokreni_homing, Home_y => "Motor_DB"."Motor_2_y-os".Pokreni_homing, Željeni_apsolutni_pomak_x => "Motor_DB"."Motor_1_x-os".Željena_pozicija, Željeni_apsolutni_pomak_y => "Motor_DB"."Motor_2_y-os".Željena_pozicija, Izvršavanje_pomaka_x => "Motor_DB"."Motor_1_x-os".Pokreni_izvršavanje_pomaka_apsolutno, Izvršavanje_pomaka_y => "Motor_DB"."Motor_2_y-os".Pokreni_izvršavanje_pomaka_apsolutno, Zaustavljanje_x => "Motor_DB"."Motor_1_x-os".Pokreni_zaustavljanje, Zaustavljanje_y => "Motor_DB"."Motor_2_y-os".Pokreni_zaustavljanje, Kraj_paletizacije => "Automatsko_upravljanje".Kraj_paletizacije)
      Contact( "Automatsko_upravljanje".Kraj_paletizacije )
      R_Coil( "Automatsko_upravljanje".Paletizacija )
   END_RUNG
   // the same network as SCL:
   "Paletizacija_DB"(EN := "Automatsko_upravljanje".Automatski_režim AND NOT "Automatsko_upravljanje".Lokalizacija_objekata_i_sortiranje,   // "Paletizacija"
                     Senzor_cilindar_uvučen := "Dist_ulaz5",
                     Senzor_cilindar_izvučen := "Dist_ulaz6",
                     Senzor_hvataljka_zatvorena := "Dist_ulaz8",
                     Senzor_hvataljka_otvorena := "Dist_ulaz7",
                     Home_izvršeno_x := "Motor_DB"."Motor_1_x-os".Home_Izvršeno,
                     Home_izvršeno_y := "Motor_DB"."Motor_2_y-os".Home_Izvršeno,
                     Trenutna_pozicija_x := "Axis_1".ActualPosition,
                     Trenutna_pozicija_y := "Axis_2".ActualPosition,
                     Pomak_izvršen_x := "Motor_DB"."Motor_1_x-os".Pomak_Apsolutno_Izvršeno,
                     Pomak_izvršen_y := "Motor_DB"."Motor_2_y-os".Pomak_Apsolutno_Izvršeno,
                     Broj_komada_palete_x := "Automatsko_upravljanje".Broj_komada_palete_x,
                     Broj_komada_palete_y := "Automatsko_upravljanje".Broj_komada_palete_y,
                     Koordinata_palete_izuzimanja_x := 10.0,
                     Koordinata_palete_izuzimanja_y := 10.0,
                     Koordinata_palete_odlaganja_x := 40.0,
                     Koordinata_palete_odlaganja_y := 70.0,
                     Pauza := "Automatsko_upravljanje".Pauza,
                     Poziv_paletizacija := "Automatsko_upravljanje".Paletizacija,
                     Aktivacija_cilindra => "Pneumatske_komponente".Aktivacija_cilindra,
                     Aktivacija_hvataljke => "Pneumatske_komponente".Aktivacija_hvataljke,
                     Home_x => "Motor_DB"."Motor_1_x-os".Pokreni_homing,
                     Home_y => "Motor_DB"."Motor_2_y-os".Pokreni_homing,
                     Željeni_apsolutni_pomak_x => "Motor_DB"."Motor_1_x-os".Željena_pozicija,
                     Željeni_apsolutni_pomak_y => "Motor_DB"."Motor_2_y-os".Željena_pozicija,
                     Izvršavanje_pomaka_x => "Motor_DB"."Motor_1_x-os".Pokreni_izvršavanje_pomaka_apsolutno,
                     Izvršavanje_pomaka_y => "Motor_DB"."Motor_2_y-os".Pokreni_izvršavanje_pomaka_apsolutno,
                     Zaustavljanje_x => "Motor_DB"."Motor_1_x-os".Pokreni_zaustavljanje,
                     Zaustavljanje_y => "Motor_DB"."Motor_2_y-os".Pokreni_zaustavljanje,
                     Kraj_paletizacije => "Automatsko_upravljanje".Kraj_paletizacije,
                     ENO => #_w1);
   IF #_w1 AND "Automatsko_upravljanje".Kraj_paletizacije THEN
       "Automatsko_upravljanje".Paletizacija := FALSE;
   END_IF;
END_REGION

REGION Network 4: TCP/IP komunikacija - slanje, primanje i obrada podataka
   // Opis koda; Komentari:
   // Tajmer za slanje poruke mora biti isključivo veći od Tajmera za primanje poruke,
   // inače će se primiti više podataka (više od samo jednog stringa), koji će ostati u
   // memoriji, te će manipulator u tom slučaju više puta odratiti istu putanju
   // 
   // Primaju se podatci u bajtovima, odnosno može se očitavati character po character iz poslanog stringa
   // Primljeni string sastoji se od x koordinate objekta u pikselima, y koordinate objekta u pikselima i broj koji određuje boju objekta
   // (npr. '812 254 0' - označava 812 pixel po x koordinati, 254 pixel po y koordinati i 0 označuje definiranu boju iz python skripte)
   // 
   // Svaki string između gore navedenih podataka ima razmak koji označava kraj jednog i početak drugog podatka, te se pomoću te informacije razdvajaju varijable u četvrtom retku
   // Character u ASCII zapisu može se izraziti u dekadskom sustavu, te broj 0 kao ASCII character ima vrijednost 48, a broj 9 kao ASCII character ima vrijednost 57 
   // (npr. character iz stringa = '0' -> kao dekadski je integer = 48 -> oduzimanjem broja 48 od charactera iz stringa dobiva se željena integer (cijelobrojna) vrijednost
   // Kako se šalje character po character, mora se prethodno dobiveni character pomnožiti sa 10 (u dekadskom sustavu) i zbrojiti s novim kako bi se dobila željena potpuna informacija o koordinatama
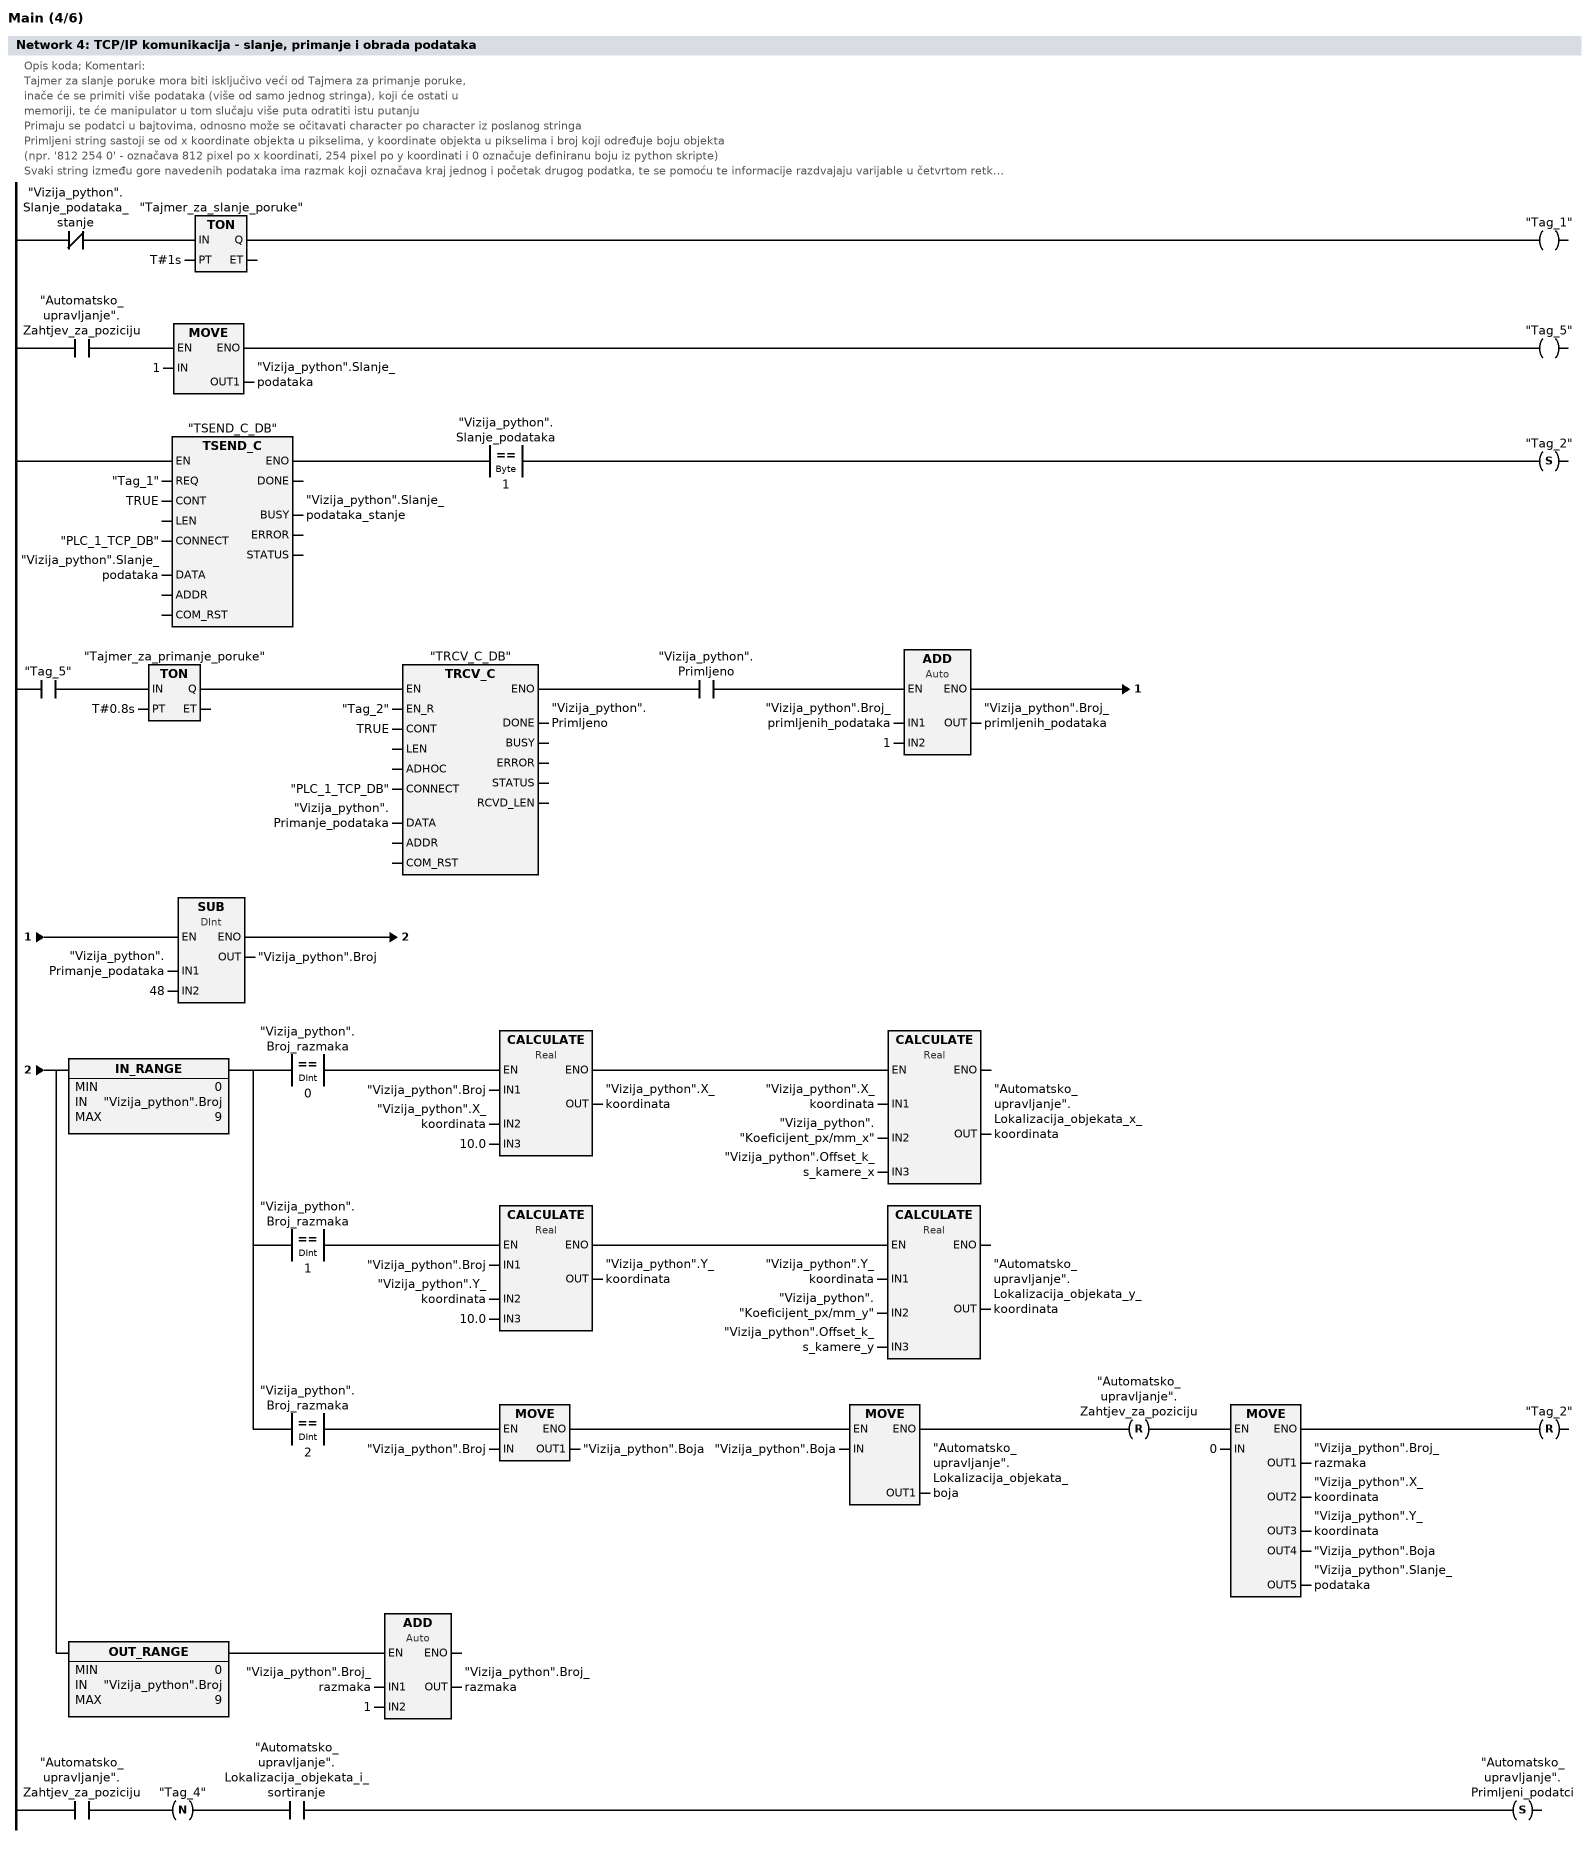
   // ENO of a box is taken as its EN; it also drops when the box reports an error
   "Tajmer_za_slanje_poruke".TON(IN := NOT "Vizija_python".Slanje_podataka_stanje, PT := T#1s);
   "Tag_1" := "Tajmer_za_slanje_poruke".Q;
   IF "Automatsko_upravljanje".Zahtjev_za_poziciju THEN "Vizija_python".Slanje_podataka := 1; END_IF;
   "Tag_5" := "Automatsko_upravljanje".Zahtjev_za_poziciju;
   "TSEND_C_DB"(REQ := "Tag_1",   // TSEND_C
                CONT := TRUE,
                CONNECT := "PLC_1_TCP_DB",
                DATA := "Vizija_python".Slanje_podataka,
                BUSY => "Vizija_python".Slanje_podataka_stanje);
   IF "Vizija_python".Slanje_podataka = 1 THEN "Tag_2" := TRUE; END_IF;
   "Tajmer_za_primanje_poruke".TON(IN := "Tag_5", PT := T#0.8s);
   #_w1 := "Tajmer_za_primanje_poruke".Q;
   IF #_w1 THEN
       "TRCV_C_DB"(EN_R := "Tag_2",   // TRCV_C
                   CONT := TRUE,
                   CONNECT := "PLC_1_TCP_DB",
                   DATA := "Vizija_python".Primanje_podataka,
                   DONE => "Vizija_python".Primljeno);
   END_IF;
   #_w2 := #_w1 AND "Vizija_python".Primljeno;
   IF #_w2 THEN
       "Vizija_python".Broj_primljenih_podataka := "Vizija_python".Broj_primljenih_podataka + 1;
       "Vizija_python".Broj := "Vizija_python".Primanje_podataka - 48;
   END_IF;
   #_w3 := #_w2 AND (0 <= "Vizija_python".Broj) AND ("Vizija_python".Broj <= 9);
   IF #_w3 AND ("Vizija_python".Broj_razmaka = 0) THEN
       "Vizija_python".X_koordinata := "Vizija_python".Broj+"Vizija_python".X_koordinata*10.0;
       "Automatsko_upravljanje".Lokalizacija_objekata_x_koordinata := "Vizija_python".X_koordinata/"Vizija_python"."Koeficijent_px/mm_x"+"Vizija_python".Offset_k_s_kamere_x;
   END_IF;
   IF #_w3 AND ("Vizija_python".Broj_razmaka = 1) THEN
       "Vizija_python".Y_koordinata := "Vizija_python".Broj+"Vizija_python".Y_koordinata*10.0;
       "Automatsko_upravljanje".Lokalizacija_objekata_y_koordinata := "Vizija_python".Y_koordinata/"Vizija_python"."Koeficijent_px/mm_y"+"Vizija_python".Offset_k_s_kamere_y;
   END_IF;
   IF #_w3 AND ("Vizija_python".Broj_razmaka = 2) THEN
       "Vizija_python".Boja := "Vizija_python".Broj;
       "Automatsko_upravljanje".Lokalizacija_objekata_boja := "Vizija_python".Boja;
       "Automatsko_upravljanje".Zahtjev_za_poziciju := FALSE;
   END_IF;
   #_w4 := #_w3 AND ("Vizija_python".Broj_razmaka = 2);
   IF #_w4 THEN
       "Vizija_python".Broj_razmaka := 0;
       "Vizija_python".X_koordinata := 0;
       "Vizija_python".Y_koordinata := 0;
       "Vizija_python".Boja := 0;
       "Vizija_python".Slanje_podataka := 0;
       "Tag_2" := FALSE;
   END_IF;
   IF #_w2 AND (("Vizija_python".Broj < 0) OR ("Vizija_python".Broj > 9)) THEN
       "Vizija_python".Broj_razmaka := "Vizija_python".Broj_razmaka + 1;
   END_IF;
   #_w5 := NOT "Automatsko_upravljanje".Zahtjev_za_poziciju AND "Tag_4";   // falling edge
   "Tag_4" := "Automatsko_upravljanje".Zahtjev_za_poziciju;
   IF #_w5 AND "Automatsko_upravljanje".Lokalizacija_objekata_i_sortiranje THEN
       "Automatsko_upravljanje".Primljeni_podatci := TRUE;
   END_IF;
END_REGION

REGION Network 5: Lokalizacija objekata
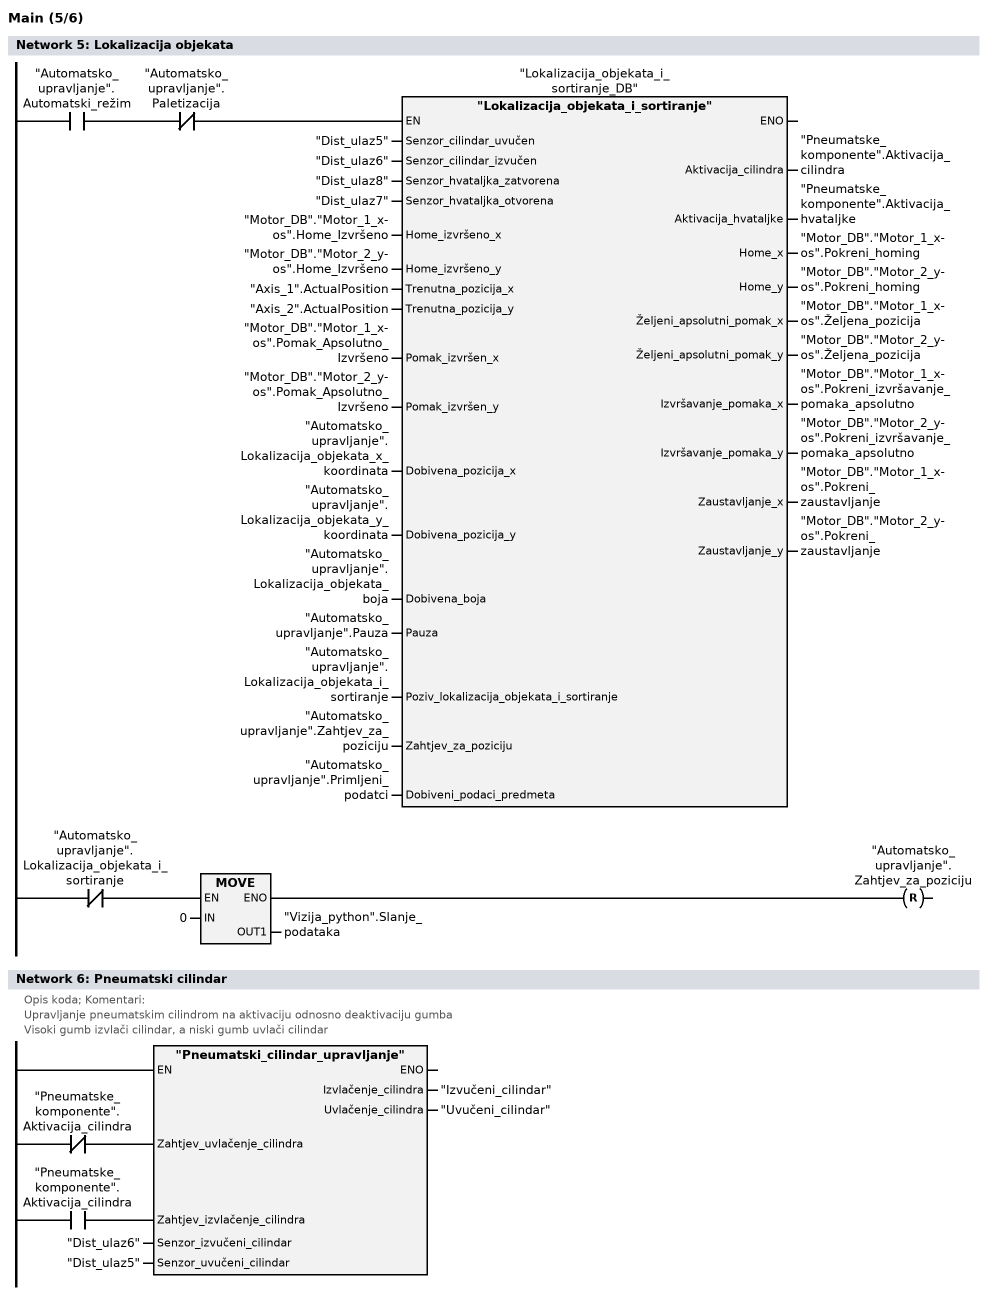
   RUNG wire#powerrail
      Contact( "Automatsko_upravljanje".Automatski_režim )
      I_Contact( "Automatsko_upravljanje".Paletizacija )
      "Lokalizacija_objekata_i_sortiranje_DB"(Senzor_cilindar_uvučen := "Dist_ulaz5", Senzor_cilindar_izvučen := "Dist_ulaz6", Senzor_hvataljka_zatvorena := "Dist_ulaz8", Senzor_hvataljka_otvorena := "Dist_ulaz7", Home_izvršeno_x := "Motor_DB"."Motor_1_x-os".Home_Izvršeno, Home_izvršeno_y := "Motor_DB"."Motor_2_y-os".Home_Izvršeno, Trenutna_pozicija_x := "Axis_1".ActualPosition, Trenutna_pozicija_y := "Axis_2".ActualPosition, Pomak_izvršen_x := "Motor_DB"."Motor_1_x-os".Pomak_Apsolutno_Izvršeno, Pomak_izvršen_y := "Motor_DB"."Motor_2_y-os".Pomak_Apsolutno_Izvršeno, Dobivena_pozicija_x := "Automatsko_upravljanje".Lokalizacija_objekata_x_koordinata, Dobivena_pozicija_y := "Automatsko_upravljanje".Lokalizacija_objekata_y_koordinata, Dobivena_boja := "Automatsko_upravljanje".Lokalizacija_objekata_boja, Pauza := "Automatsko_upravljanje".Pauza, Poziv_lokalizacija_objekata_i_sortiranje := "Automatsko_upravljanje".Lokalizacija_objekata_i_sortiranje, Zahtjev_za_poziciju := "Automatsko_upravljanje".Zahtjev_za_poziciju, Dobiveni_podaci_predmeta := "Automatsko_upravljanje".Primljeni_podatci, Aktivacija_cilindra => "Pneumatske_komponente".Aktivacija_cilindra, Aktivacija_hvataljke => "Pneumatske_komponente".Aktivacija_hvataljke, Home_x => "Motor_DB"."Motor_1_x-os".Pokreni_homing, Home_y => "Motor_DB"."Motor_2_y-os".Pokreni_homing, Željeni_apsolutni_pomak_x => "Motor_DB"."Motor_1_x-os".Željena_pozicija, Željeni_apsolutni_pomak_y => "Motor_DB"."Motor_2_y-os".Željena_pozicija, Izvršavanje_pomaka_x => "Motor_DB"."Motor_1_x-os".Pokreni_izvršavanje_pomaka_apsolutno, Izvršavanje_pomaka_y => "Motor_DB"."Motor_2_y-os".Pokreni_izvršavanje_pomaka_apsolutno, Zaustavljanje_x => "Motor_DB"."Motor_1_x-os".Pokreni_zaustavljanje, Zaustavljanje_y => "Motor_DB"."Motor_2_y-os".Pokreni_zaustavljanje)
   END_RUNG
   RUNG wire#powerrail
      I_Contact( "Automatsko_upravljanje".Lokalizacija_objekata_i_sortiranje )
      Move(in := 0, out1 => "Vizija_python".Slanje_podataka)
      R_Coil( "Automatsko_upravljanje".Zahtjev_za_poziciju )
   END_RUNG
   // the same network as SCL:
   IF "Automatsko_upravljanje".Automatski_režim AND NOT "Automatsko_upravljanje".Paletizacija THEN
       "Lokalizacija_objekata_i_sortiranje_DB"(Senzor_cilindar_uvučen := "Dist_ulaz5",   // "Lokalizacija_objekata_i_sortiranje"
                               Senzor_cilindar_izvučen := "Dist_ulaz6",
                               Senzor_hvataljka_zatvorena := "Dist_ulaz8",
                               Senzor_hvataljka_otvorena := "Dist_ulaz7",
                               Home_izvršeno_x := "Motor_DB"."Motor_1_x-os".Home_Izvršeno,
                               Home_izvršeno_y := "Motor_DB"."Motor_2_y-os".Home_Izvršeno,
                               Trenutna_pozicija_x := "Axis_1".ActualPosition,
                               Trenutna_pozicija_y := "Axis_2".ActualPosition,
                               Pomak_izvršen_x := "Motor_DB"."Motor_1_x-os".Pomak_Apsolutno_Izvršeno,
                               Pomak_izvršen_y := "Motor_DB"."Motor_2_y-os".Pomak_Apsolutno_Izvršeno,
                               Dobivena_pozicija_x := "Automatsko_upravljanje".Lokalizacija_objekata_x_koordinata,
                               Dobivena_pozicija_y := "Automatsko_upravljanje".Lokalizacija_objekata_y_koordinata,
                               Dobivena_boja := "Automatsko_upravljanje".Lokalizacija_objekata_boja,
                               Pauza := "Automatsko_upravljanje".Pauza,
                               Poziv_lokalizacija_objekata_i_sortiranje := "Automatsko_upravljanje".Lokalizacija_objekata_i_sortiranje,
                               Zahtjev_za_poziciju := "Automatsko_upravljanje".Zahtjev_za_poziciju,
                               Dobiveni_podaci_predmeta := "Automatsko_upravljanje".Primljeni_podatci,
                               Aktivacija_cilindra => "Pneumatske_komponente".Aktivacija_cilindra,
                               Aktivacija_hvataljke => "Pneumatske_komponente".Aktivacija_hvataljke,
                               Home_x => "Motor_DB"."Motor_1_x-os".Pokreni_homing,
                               Home_y => "Motor_DB"."Motor_2_y-os".Pokreni_homing,
                               Željeni_apsolutni_pomak_x => "Motor_DB"."Motor_1_x-os".Željena_pozicija,
                               Željeni_apsolutni_pomak_y => "Motor_DB"."Motor_2_y-os".Željena_pozicija,
                               Izvršavanje_pomaka_x => "Motor_DB"."Motor_1_x-os".Pokreni_izvršavanje_pomaka_apsolutno,
                               Izvršavanje_pomaka_y => "Motor_DB"."Motor_2_y-os".Pokreni_izvršavanje_pomaka_apsolutno,
                               Zaustavljanje_x => "Motor_DB"."Motor_1_x-os".Pokreni_zaustavljanje,
                               Zaustavljanje_y => "Motor_DB"."Motor_2_y-os".Pokreni_zaustavljanje);
   END_IF;
   IF NOT "Automatsko_upravljanje".Lokalizacija_objekata_i_sortiranje THEN
       "Vizija_python".Slanje_podataka := 0;
       "Automatsko_upravljanje".Zahtjev_za_poziciju := FALSE;
   END_IF;
END_REGION

REGION Network 6: Pneumatski cilindar
   // Opis koda; Komentari:
   // Upravljanje pneumatskim cilindrom na aktivaciju odnosno deaktivaciju gumba
   // Visoki gumb izvlači cilindar, a niski gumb uvlači cilindar
   RUNG wire#powerrail
      "Pneumatski_cilindar_upravljanje"(Zahtjev_uvlačenje_cilindra := wire#w1, Zahtjev_izvlačenje_cilindra := wire#w2, Senzor_izvučeni_cilindar := "Dist_ulaz6", Senzor_uvučeni_cilindar := "Dist_ulaz5", Izvlačenje_cilindra => "Izvučeni_cilindar", Uvlačenje_cilindra => "Uvučeni_cilindar")
   END_RUNG
   RUNG wire#powerrail
      I_Contact( "Pneumatske_komponente".Aktivacija_cilindra )
   END_RUNG wire#w1
   RUNG wire#powerrail
      Contact( "Pneumatske_komponente".Aktivacija_cilindra )
   END_RUNG wire#w2
   // the same network as SCL:
   "Pneumatski_cilindar_upravljanje"(Zahtjev_uvlačenje_cilindra := NOT "Pneumatske_komponente".Aktivacija_cilindra,
                           Zahtjev_izvlačenje_cilindra := "Pneumatske_komponente".Aktivacija_cilindra,
                           Senzor_izvučeni_cilindar := "Dist_ulaz6",
                           Senzor_uvučeni_cilindar := "Dist_ulaz5",
                           Izvlačenje_cilindra => "Izvučeni_cilindar",
                           Uvlačenje_cilindra => "Uvučeni_cilindar");
END_REGION

REGION Network 7: Pnneumatska hvataljka
   // Oppis koda; Komentari:
   // Upravljanje pneumatskom hvataljkom na aktivaciju odnosno deaktivaciju gumba
   // Visoki gumb zatvara hvataljku, a niski gumb otvara hvataljku
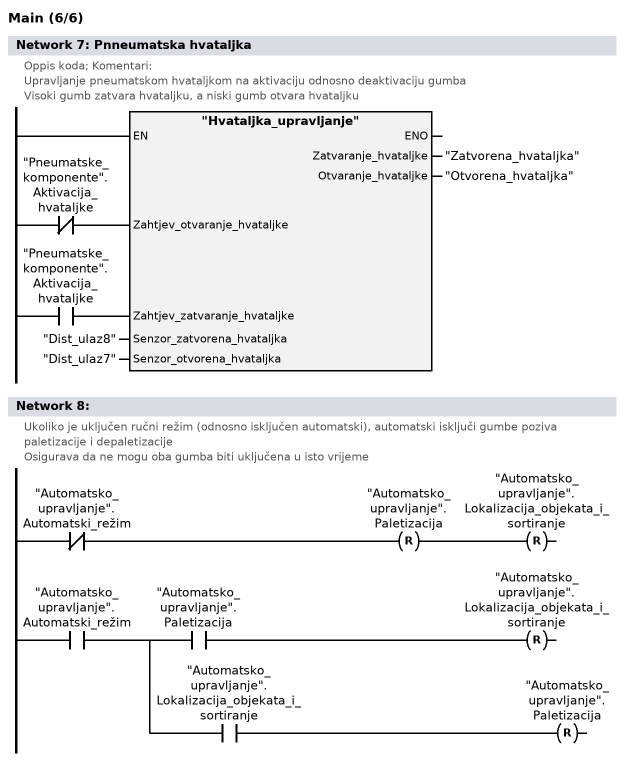
   RUNG wire#powerrail
      "Hvataljka_upravljanje"(Zahtjev_otvaranje_hvataljke := wire#w1, Zahtjev_zatvaranje_hvataljke := wire#w2, Senzor_zatvorena_hvataljka := "Dist_ulaz8", Senzor_otvorena_hvataljka := "Dist_ulaz7", Zatvaranje_hvataljke => "Zatvorena_hvataljka", Otvaranje_hvataljke => "Otvorena_hvataljka")
   END_RUNG
   RUNG wire#powerrail
      I_Contact( "Pneumatske_komponente".Aktivacija_hvataljke )
   END_RUNG wire#w1
   RUNG wire#powerrail
      Contact( "Pneumatske_komponente".Aktivacija_hvataljke )
   END_RUNG wire#w2
   // the same network as SCL:
   "Hvataljka_upravljanje"(Zahtjev_otvaranje_hvataljke := NOT "Pneumatske_komponente".Aktivacija_hvataljke,
                           Zahtjev_zatvaranje_hvataljke := "Pneumatske_komponente".Aktivacija_hvataljke,
                           Senzor_zatvorena_hvataljka := "Dist_ulaz8",
                           Senzor_otvorena_hvataljka := "Dist_ulaz7",
                           Zatvaranje_hvataljke => "Zatvorena_hvataljka",
                           Otvaranje_hvataljke => "Otvorena_hvataljka");
END_REGION

REGION Network 8
   // Ukoliko je uključen ručni režim (odnosno isključen automatski), automatski isključi gumbe poziva paletizacije i depaletizacije
   // Osigurava da ne mogu oba gumba biti uključena u isto vrijeme
   RUNG wire#powerrail
      I_Contact( "Automatsko_upravljanje".Automatski_režim )
      R_Coil( "Automatsko_upravljanje".Paletizacija )
      R_Coil( "Automatsko_upravljanje".Lokalizacija_objekata_i_sortiranje )
   END_RUNG
   RUNG wire#powerrail
      Contact( "Automatsko_upravljanje".Automatski_režim )
      wire#w1
      Contact( "Automatsko_upravljanje".Paletizacija )
      R_Coil( "Automatsko_upravljanje".Lokalizacija_objekata_i_sortiranje )
   END_RUNG
   RUNG wire#w1
      Contact( "Automatsko_upravljanje".Lokalizacija_objekata_i_sortiranje )
      R_Coil( "Automatsko_upravljanje".Paletizacija )
   END_RUNG
   // the same network as SCL:
   IF NOT "Automatsko_upravljanje".Automatski_režim THEN
       "Automatsko_upravljanje".Paletizacija := FALSE;
       "Automatsko_upravljanje".Lokalizacija_objekata_i_sortiranje := FALSE;
   END_IF;
   IF "Automatsko_upravljanje".Automatski_režim AND "Automatsko_upravljanje".Paletizacija THEN
       "Automatsko_upravljanje".Lokalizacija_objekata_i_sortiranje := FALSE;
   END_IF;
   IF "Automatsko_upravljanje".Automatski_režim AND "Automatsko_upravljanje".Lokalizacija_objekata_i_sortiranje THEN
       "Automatsko_upravljanje".Paletizacija := FALSE;
   END_IF;
END_REGION
END_ORGANIZATION_BLOCK

(* ===== HMI "HMI_RT_1" =====
system functions are stored by id; their names below are inferred from use
connection "HMI_Connection_1": ETHERNET, SMART_S7_1200_OMS

HMI tags "Default tag table"
   "Motor_DB_Motor_1_x-os_Uključi_motor" : Bool = PLC Motor_DB.Motor_1_x-os.Uključi_motor, 100 ms
   "Motor_DB_Motor_1_x-os_Trenutna_pozicija" : Real = PLC Motor_DB.Motor_1_x-os.Trenutna_pozicija, 100 ms
   "Motor_DB_Motor_2_y-os_Trenutna_pozicija" : Real = PLC Motor_DB.Motor_2_y-os.Trenutna_pozicija, 100 ms
   "Motor_DB_Motor_1_x-os_Power_Status" : Bool = PLC Motor_DB.Motor_1_x-os.Power_Status, 100 ms
   "Motor_DB_Motor_2_y-os_Power_Status" : Bool = PLC Motor_DB.Motor_2_y-os.Power_Status, 100 ms
   "Motor_DB_Motor_2_y-os_Uključi_motor" : Bool = PLC Motor_DB.Motor_2_y-os.Uključi_motor, 100 ms
   "Motor_DB_Motor_1_x-os_Pokreni_homing" : Bool = PLC Motor_DB.Motor_1_x-os.Pokreni_homing, 100 ms
   "Motor_DB_Motor_2_y-os_Pokreni_homing" : Bool = PLC Motor_DB.Motor_2_y-os.Pokreni_homing, 100 ms
   "Motor_DB_Motor_2_y-os_Potvrdi_error(reset)" : Bool = PLC Motor_DB.Motor_2_y-os.Potvrdi_error(reset), 100 ms
   "Motor_DB_Motor_1_x-os_Potvrdi_error(reset)" : Bool = PLC Motor_DB.Motor_1_x-os.Potvrdi_error(reset), 100 ms
   "Motor_DB_Motor_1_x-os_Pokreni_zaustavljanje" : Bool = PLC Motor_DB.Motor_1_x-os.Pokreni_zaustavljanje, 100 ms
   "Motor_DB_Motor_2_y-os_Pokreni_zaustavljanje" : Bool = PLC Motor_DB.Motor_2_y-os.Pokreni_zaustavljanje, 100 ms
   "Motor_DB_Motor_1_x-os_Pokreni_izvršavanje_pomaka_apsolutno" : Bool = PLC Motor_DB.Motor_1_x-os.Pokreni_izvršavanje_pomaka_apsolutno, 100 ms
   "Motor_DB_Motor_2_y-os_Pokreni_izvršavanje_pomaka_apsolutno" : Bool = PLC Motor_DB.Motor_2_y-os.Pokreni_izvršavanje_pomaka_apsolutno, 100 ms
   "Motor_DB_Motor_2_y-os_Željena_pozicija" : Real = PLC Motor_DB.Motor_2_y-os.Željena_pozicija, 100 ms
   "Motor_DB_Motor_1_x-os_Željena_pozicija" : Real = PLC Motor_DB.Motor_1_x-os.Željena_pozicija, 100 ms
   "Motor_DB_Motor_1_x-os_Željeni_pomak" : Real = PLC Motor_DB.Motor_1_x-os.Željeni_pomak, 100 ms
   "Motor_DB_Motor_2_y-os_Željeni_pomak" : Real = PLC Motor_DB.Motor_2_y-os.Željeni_pomak, 100 ms
   "Motor_DB_Motor_2_y-os_Pokreni_izvršavanje_pomaka_relativno" : Bool = PLC Motor_DB.Motor_2_y-os.Pokreni_izvršavanje_pomaka_relativno, 100 ms
   "Motor_DB_Motor_1_x-os_Pokreni_izvršavanje_pomaka_relativno" : Bool = PLC Motor_DB.Motor_1_x-os.Pokreni_izvršavanje_pomaka_relativno, 100 ms
   "Rucno_upravljanje_LIJEVO" : Bool = PLC Rucno_upravljanje.LIJEVO, 100 ms
   "Rucno_upravljanje_GORE" : Bool = PLC Rucno_upravljanje.GORE, 100 ms
   "Rucno_upravljanje_DESNO" : Bool = PLC Rucno_upravljanje.DESNO, 100 ms
   "Rucno_upravljanje_DOLJE" : Bool = PLC Rucno_upravljanje.DOLJE, 100 ms
   "Rucno_upravljanje_GD_brzina" : Real = PLC Rucno_upravljanje.GD_brzina, 100 ms
   "Rucno_upravljanje_LD_brzina" : Real = PLC Rucno_upravljanje.LD_brzina, 100 ms
   "Izvučeni_cilindar" : Bool = PLC Zatvorena_hvataljka AT %Q4.5, 100 ms
   "Pneumatske_komponente_Aktivacija_cilindra" : Bool = PLC Pneumatske_komponente.Aktivacija_cilindra, 100 ms
   "Pneumatske_komponente_Aktivacija_hvataljke" : Bool = PLC Pneumatske_komponente.Aktivacija_hvataljke, 100 ms
   "Dist_ulaz5" : Bool = PLC Dist_ulaz5 AT %I2.4, 100 ms
   "Dist_ulaz7" : Bool = PLC Dist_ulaz7 AT %I2.6, 100 ms
   "Automatsko_upravljanje_Automatski_režim" : Bool = PLC Automatsko_upravljanje.Automatski_režim, 100 ms
   "Automatsko_upravljanje_Paletizacija" : Bool = PLC Automatsko_upravljanje.Paletizacija, 100 ms
   "Automatsko_upravljanje_Broj_komada_palete_y" : Int = PLC Automatsko_upravljanje.Broj_komada_palete_y, 100 ms
   "Automatsko_upravljanje_Broj_komada_palete_x" : Int = PLC Automatsko_upravljanje.Broj_komada_palete_x, 100 ms
   "Automatsko_upravljanje_Pauza" : Bool = PLC Automatsko_upravljanje.Pauza, 100 ms
   "Automatsko_upravljanje_Lokalizacija_objekata" : Bool = PLC Automatsko_upravljanje.Lokalizacija_objekata_i_sortiranje, 100 ms

text list "Axis_1_Power_Status": 0 'OFF'; 1 'ON'

text list "Axis_2_Power_Status": 0 'OFF'; 1 'ON'

text list "Stanje_cilindra": 0 'Cilindar izvučen'; 1 'Cilindar uvučen'

text list "Stanje_hvataljke": 0 'Hvataljka zatvorena'; 1 'Hvataljka otvorena'

text list "Broj_komada_u_paleti_x-os": 1 '1'; 2 '2'; 3 '3'; 4 '4'

text list "Broj_komada_u_paleti_y-os": 1 '1'; 2 '2'; 3 '3'

